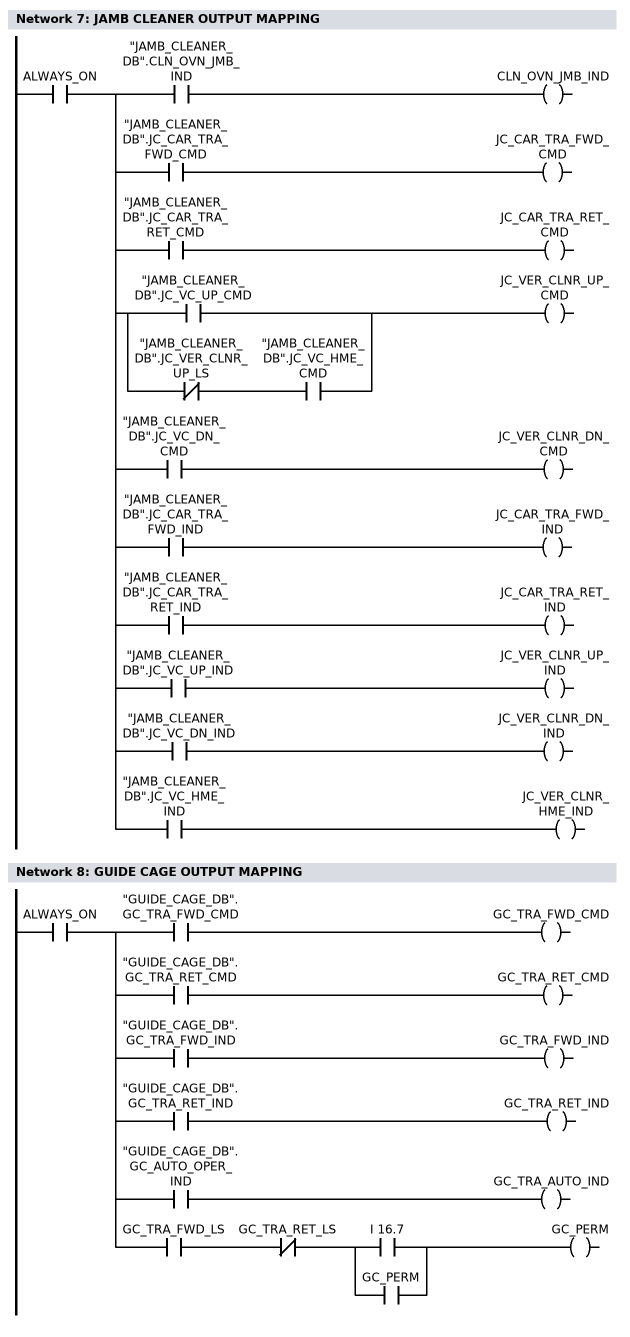
[picture p24: OUTPUT_MAPPING networks 7-8]
NETWORK
TITLE = JAMB CLEANER OUTPUT MAPPING
//JAMB CLEANER 
//
      A     "ALWAYS_ON";
      =     L 0.0;
      A     L 0.0;
      A     "JAMB_CLEANER_DB".CLN_OVN_JMB_IND;
      =     "CLN_OVN_JMB_IND";
      A     L 0.0;
      A     "JAMB_CLEANER_DB".JC_CAR_TRA_FWD_CMD;
      =     "JC_CAR_TRA_FWD_CMD";
      A     L 0.0;
      A     "JAMB_CLEANER_DB".JC_CAR_TRA_RET_CMD;
      =     "JC_CAR_TRA_RET_CMD";
      A     L 0.0;
      A(;
      O     "JAMB_CLEANER_DB".JC_VC_UP_CMD;
      O;
      AN    "JAMB_CLEANER_DB".JC_VER_CLNR_UP_LS;
      A     "JAMB_CLEANER_DB".JC_VC_HME_CMD;
      );
      =     "JC_VER_CLNR_UP_CMD";
      A     L 0.0;
      A     "JAMB_CLEANER_DB".JC_VC_DN_CMD;
      =     "JC_VER_CLNR_DN_CMD";
      A     L 0.0;
      A     "JAMB_CLEANER_DB".JC_CAR_TRA_FWD_IND;
      =     "JC_CAR_TRA_FWD_IND";
      A     L 0.0;
      A     "JAMB_CLEANER_DB".JC_CAR_TRA_RET_IND;
      =     "JC_CAR_TRA_RET_IND";
      A     L 0.0;
      A     "JAMB_CLEANER_DB".JC_VC_UP_IND;
      =     "JC_VER_CLNR_UP_IND";
      A     L 0.0;
      A     "JAMB_CLEANER_DB".JC_VC_DN_IND;
      =     "JC_VER_CLNR_DN_IND";
      A     L 0.0;
      A     "JAMB_CLEANER_DB".JC_VC_HME_IND;
      =     "JC_VER_CLNR_HME_IND";
NETWORK
TITLE = GUIDE CAGE OUTPUT MAPPING
      A     "ALWAYS_ON";
      =     L 0.0;
      A     L 0.0;
      A     "GUIDE_CAGE_DB".GC_TRA_FWD_CMD;
      =     "GC_TRA_FWD_CMD";
      A     L 0.0;
      A     "GUIDE_CAGE_DB".GC_TRA_RET_CMD;
      =     "GC_TRA_RET_CMD";
      A     L 0.0;
      A     "GUIDE_CAGE_DB".GC_TRA_FWD_IND;
      =     "GC_TRA_FWD_IND";
      A     L 0.0;
      A     "GUIDE_CAGE_DB".GC_TRA_RET_IND;
      =     "GC_TRA_RET_IND";
      A     L 0.0;
      A     "GUIDE_CAGE_DB".GC_AUTO_OPER_IND;
      =     "GC_TRA_AUTO_IND";
      A     L 0.0;
      A     "GC_TRA_FWD_LS";
      AN    "GC_TRA_RET_LS";
      A(;
      O     I 16.7;
      O     "GC_PERM";
      );
      =     "GC_PERM";
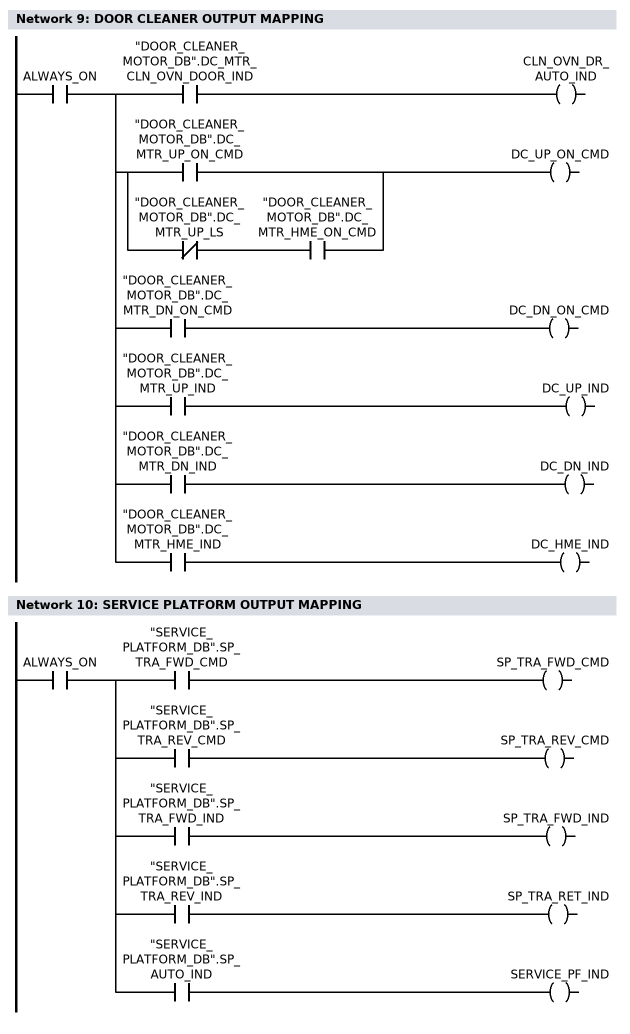
NETWORK
TITLE = DOOR CLEANER OUTPUT MAPPING
      A     "ALWAYS_ON";
      =     L 0.0;
      A     L 0.0;
      A     "DOOR_CLEANER_MOTOR_DB".DC_MTR_CLN_OVN_DOOR_IND;
      =     "CLN_OVN_DR_AUTO_IND";
      A     L 0.0;
      A(;
      O     "DOOR_CLEANER_MOTOR_DB".DC_MTR_UP_ON_CMD;
      O;
      AN    "DOOR_CLEANER_MOTOR_DB".DC_MTR_UP_LS;
      A     "DOOR_CLEANER_MOTOR_DB".DC_MTR_HME_ON_CMD;
      );
      =     "DC_UP_ON_CMD";
      A     L 0.0;
      A     "DOOR_CLEANER_MOTOR_DB".DC_MTR_DN_ON_CMD;
      =     "DC_DN_ON_CMD";
      A     L 0.0;
      A     "DOOR_CLEANER_MOTOR_DB".DC_MTR_UP_IND;
      =     "DC_UP_IND";
      A     L 0.0;
      A     "DOOR_CLEANER_MOTOR_DB".DC_MTR_DN_IND;
      =     "DC_DN_IND";
      A     L 0.0;
      A     "DOOR_CLEANER_MOTOR_DB".DC_MTR_HME_IND;
      =     "DC_HME_IND";
NETWORK
TITLE = SERVICE PLATFORM OUTPUT MAPPING
      A     "ALWAYS_ON";
      =     L 0.0;
      A     L 0.0;
      A     "SERVICE_PLATFORM_DB".SP_TRA_FWD_CMD;
      =     "SP_TRA_FWD_CMD";
      A     L 0.0;
      A     "SERVICE_PLATFORM_DB".SP_TRA_REV_CMD;
      =     "SP_TRA_REV_CMD";
      A     L 0.0;
      A     "SERVICE_PLATFORM_DB".SP_TRA_FWD_IND;
      =     "SP_TRA_FWD_IND";
      A     L 0.0;
      A     "SERVICE_PLATFORM_DB".SP_TRA_REV_IND;
      =     "SP_TRA_RET_IND";
      A     L 0.0;
      A     "SERVICE_PLATFORM_DB".SP_AUTO_IND;
      =     "SERVICE_PF_IND";
END_FUNCTION

FUNCTION "MAIN_POWER" : VOID	// FC 3
AUTHOR : Kamillas
VERSION : 0.1
BEGIN
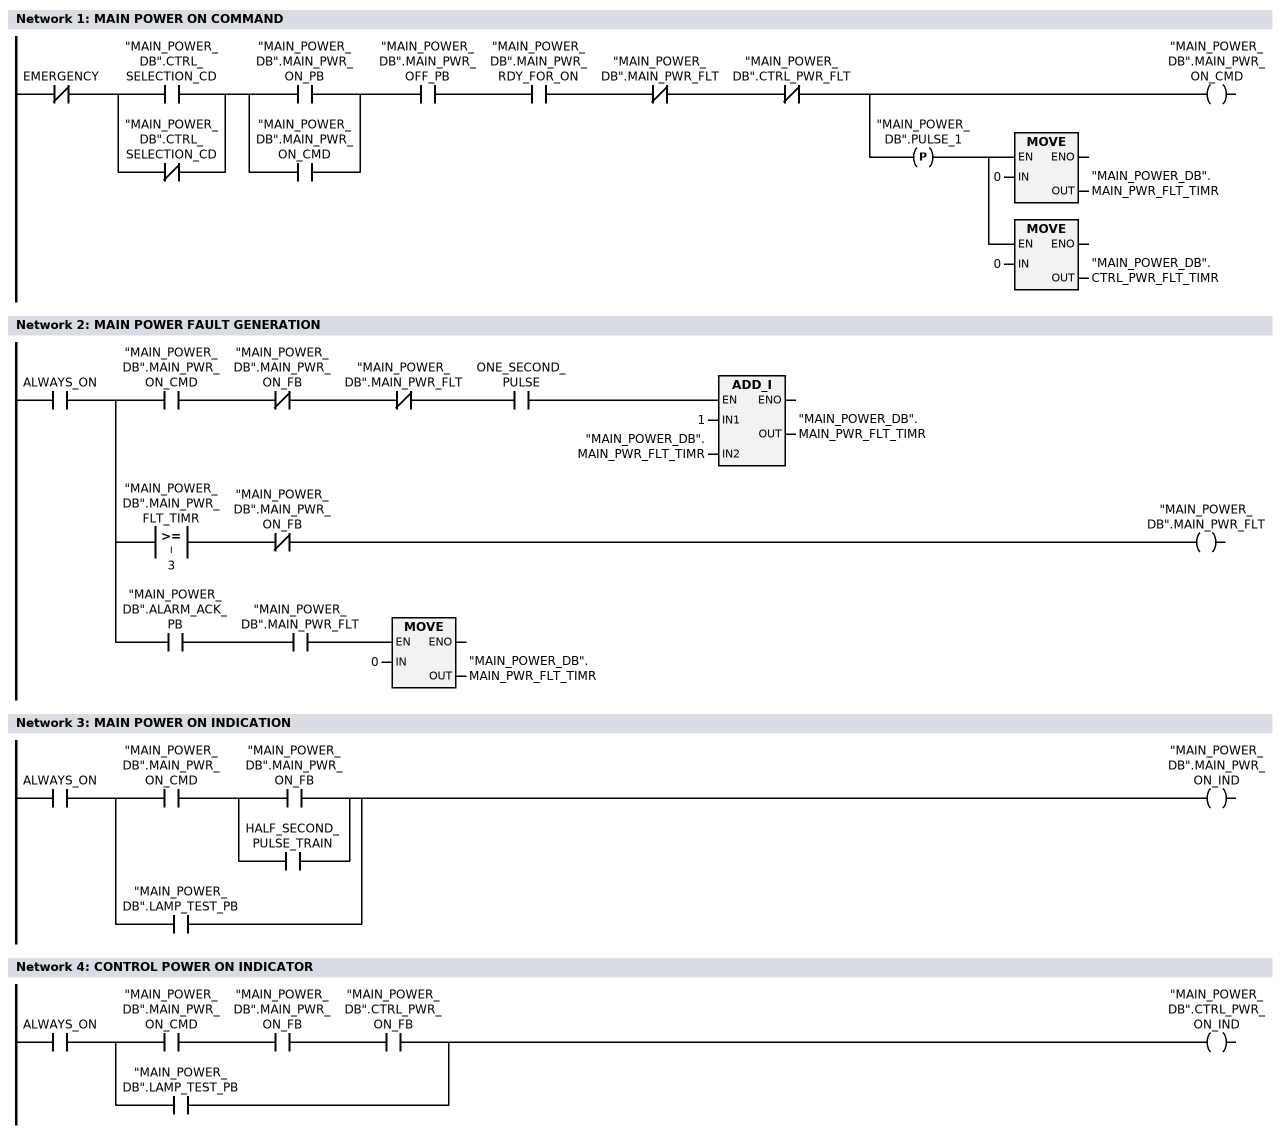
NETWORK
TITLE = MAIN POWER ON COMMAND
      AN    "EMERGENCY";
      A(;
      O     "MAIN_POWER_DB".CTRL_SELECTION_CD;
      ON    "MAIN_POWER_DB".CTRL_SELECTION_CD;
      );
      A(;
      O     "MAIN_POWER_DB".MAIN_PWR_ON_PB;
      O     "MAIN_POWER_DB".MAIN_PWR_ON_CMD;
      );
      A     "MAIN_POWER_DB".MAIN_PWR_OFF_PB;
      A     "MAIN_POWER_DB".MAIN_PWR_RDY_FOR_ON;
      AN    "MAIN_POWER_DB".MAIN_PWR_FLT;
      AN    "MAIN_POWER_DB".CTRL_PWR_FLT;
      =     L 0.0;
      A     L 0.0;
      BLD   102;
      =     "MAIN_POWER_DB".MAIN_PWR_ON_CMD;
      A     L 0.0;
      FP    "MAIN_POWER_DB".PULSE_1;
      =     L 0.1;
      A     L 0.1;
      JNB   _001;
      L     0;
      T     "MAIN_POWER_DB".MAIN_PWR_FLT_TIMR;
_001: NOP   0;
      A     L 0.1;
      JNB   _002;
      L     0;
      T     "MAIN_POWER_DB".CTRL_PWR_FLT_TIMR;
_002: NOP   0;
NETWORK
TITLE = MAIN POWER FAULT GENERATION
      A     "ALWAYS_ON";
      =     L 0.0;
      A     L 0.0;
      A     "MAIN_POWER_DB".MAIN_PWR_ON_CMD;
      AN    "MAIN_POWER_DB".MAIN_PWR_ON_FB;
      AN    "MAIN_POWER_DB".MAIN_PWR_FLT;
      A     "ONE_SECOND_PULSE";
      JNB   _003;
      L     1;
      L     "MAIN_POWER_DB".MAIN_PWR_FLT_TIMR;
      +I;
      T     "MAIN_POWER_DB".MAIN_PWR_FLT_TIMR;
_003: NOP   0;
      A     L 0.0;
      A(;
      L     "MAIN_POWER_DB".MAIN_PWR_FLT_TIMR;
      L     3;
      >=I;
      );
      AN    "MAIN_POWER_DB".MAIN_PWR_ON_FB;
      =     "MAIN_POWER_DB".MAIN_PWR_FLT;
      A     L 0.0;
      A     "MAIN_POWER_DB".ALARM_ACK_PB;
      A     "MAIN_POWER_DB".MAIN_PWR_FLT;
      JNB   _004;
      L     0;
      T     "MAIN_POWER_DB".MAIN_PWR_FLT_TIMR;
_004: NOP   0;
NETWORK
TITLE = MAIN POWER ON INDICATION
      A     "ALWAYS_ON";
      A(;
      A     "MAIN_POWER_DB".MAIN_PWR_ON_CMD;
      A(;
      O     "MAIN_POWER_DB".MAIN_PWR_ON_FB;
      O     "HALF_SECOND_PULSE_TRAIN";
      );
      O     "MAIN_POWER_DB".LAMP_TEST_PB;
      );
      =     "MAIN_POWER_DB".MAIN_PWR_ON_IND;
NETWORK
TITLE = CONTROL POWER ON INDICATOR
      A     "ALWAYS_ON";
      A(;
      A     "MAIN_POWER_DB".MAIN_PWR_ON_CMD;
      A     "MAIN_POWER_DB".MAIN_PWR_ON_FB;
      A     "MAIN_POWER_DB".CTRL_PWR_ON_FB;
      O     "MAIN_POWER_DB".LAMP_TEST_PB;
      );
      =     "MAIN_POWER_DB".CTRL_PWR_ON_IND;
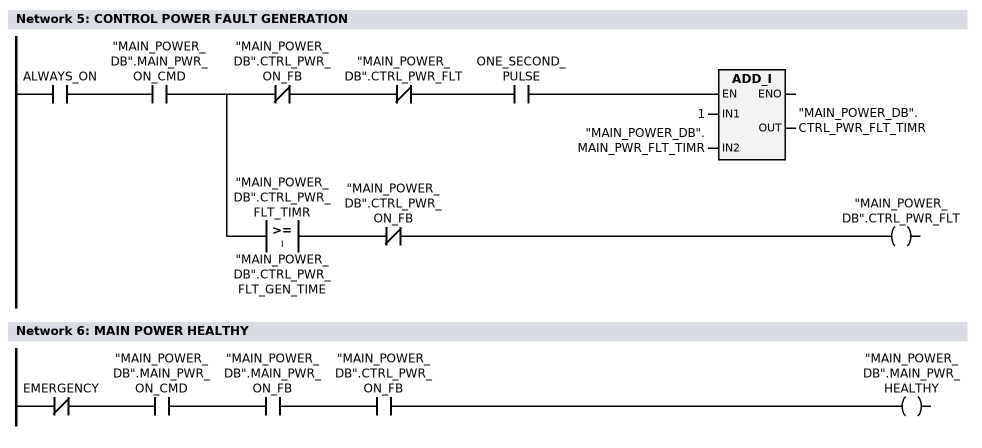
NETWORK
TITLE = CONTROL POWER FAULT GENERATION
      A     "ALWAYS_ON";
      A     "MAIN_POWER_DB".MAIN_PWR_ON_CMD;
      =     L 0.0;
      A     L 0.0;
      AN    "MAIN_POWER_DB".CTRL_PWR_ON_FB;
      AN    "MAIN_POWER_DB".CTRL_PWR_FLT;
      A     "ONE_SECOND_PULSE";
      JNB   _005;
      L     1;
      L     "MAIN_POWER_DB".MAIN_PWR_FLT_TIMR;
      +I;
      T     "MAIN_POWER_DB".CTRL_PWR_FLT_TIMR;
_005: NOP   0;
      A     L 0.0;
      A(;
      L     "MAIN_POWER_DB".CTRL_PWR_FLT_TIMR;
      L     "MAIN_POWER_DB".CTRL_PWR_FLT_GEN_TIME;
      >=I;
      );
      AN    "MAIN_POWER_DB".CTRL_PWR_ON_FB;
      =     "MAIN_POWER_DB".CTRL_PWR_FLT;
NETWORK
TITLE = MAIN POWER HEALTHY 
      AN    "EMERGENCY";
      A     "MAIN_POWER_DB".MAIN_PWR_ON_CMD;
      A     "MAIN_POWER_DB".MAIN_PWR_ON_FB;
      A     "MAIN_POWER_DB".CTRL_PWR_ON_FB;
      =     "MAIN_POWER_DB".MAIN_PWR_HEALTHY;
END_FUNCTION

FUNCTION "HYDRAULIC_SYSTEM" : VOID	// FC 4
AUTHOR : Kamillas
VERSION : 0.1
BEGIN
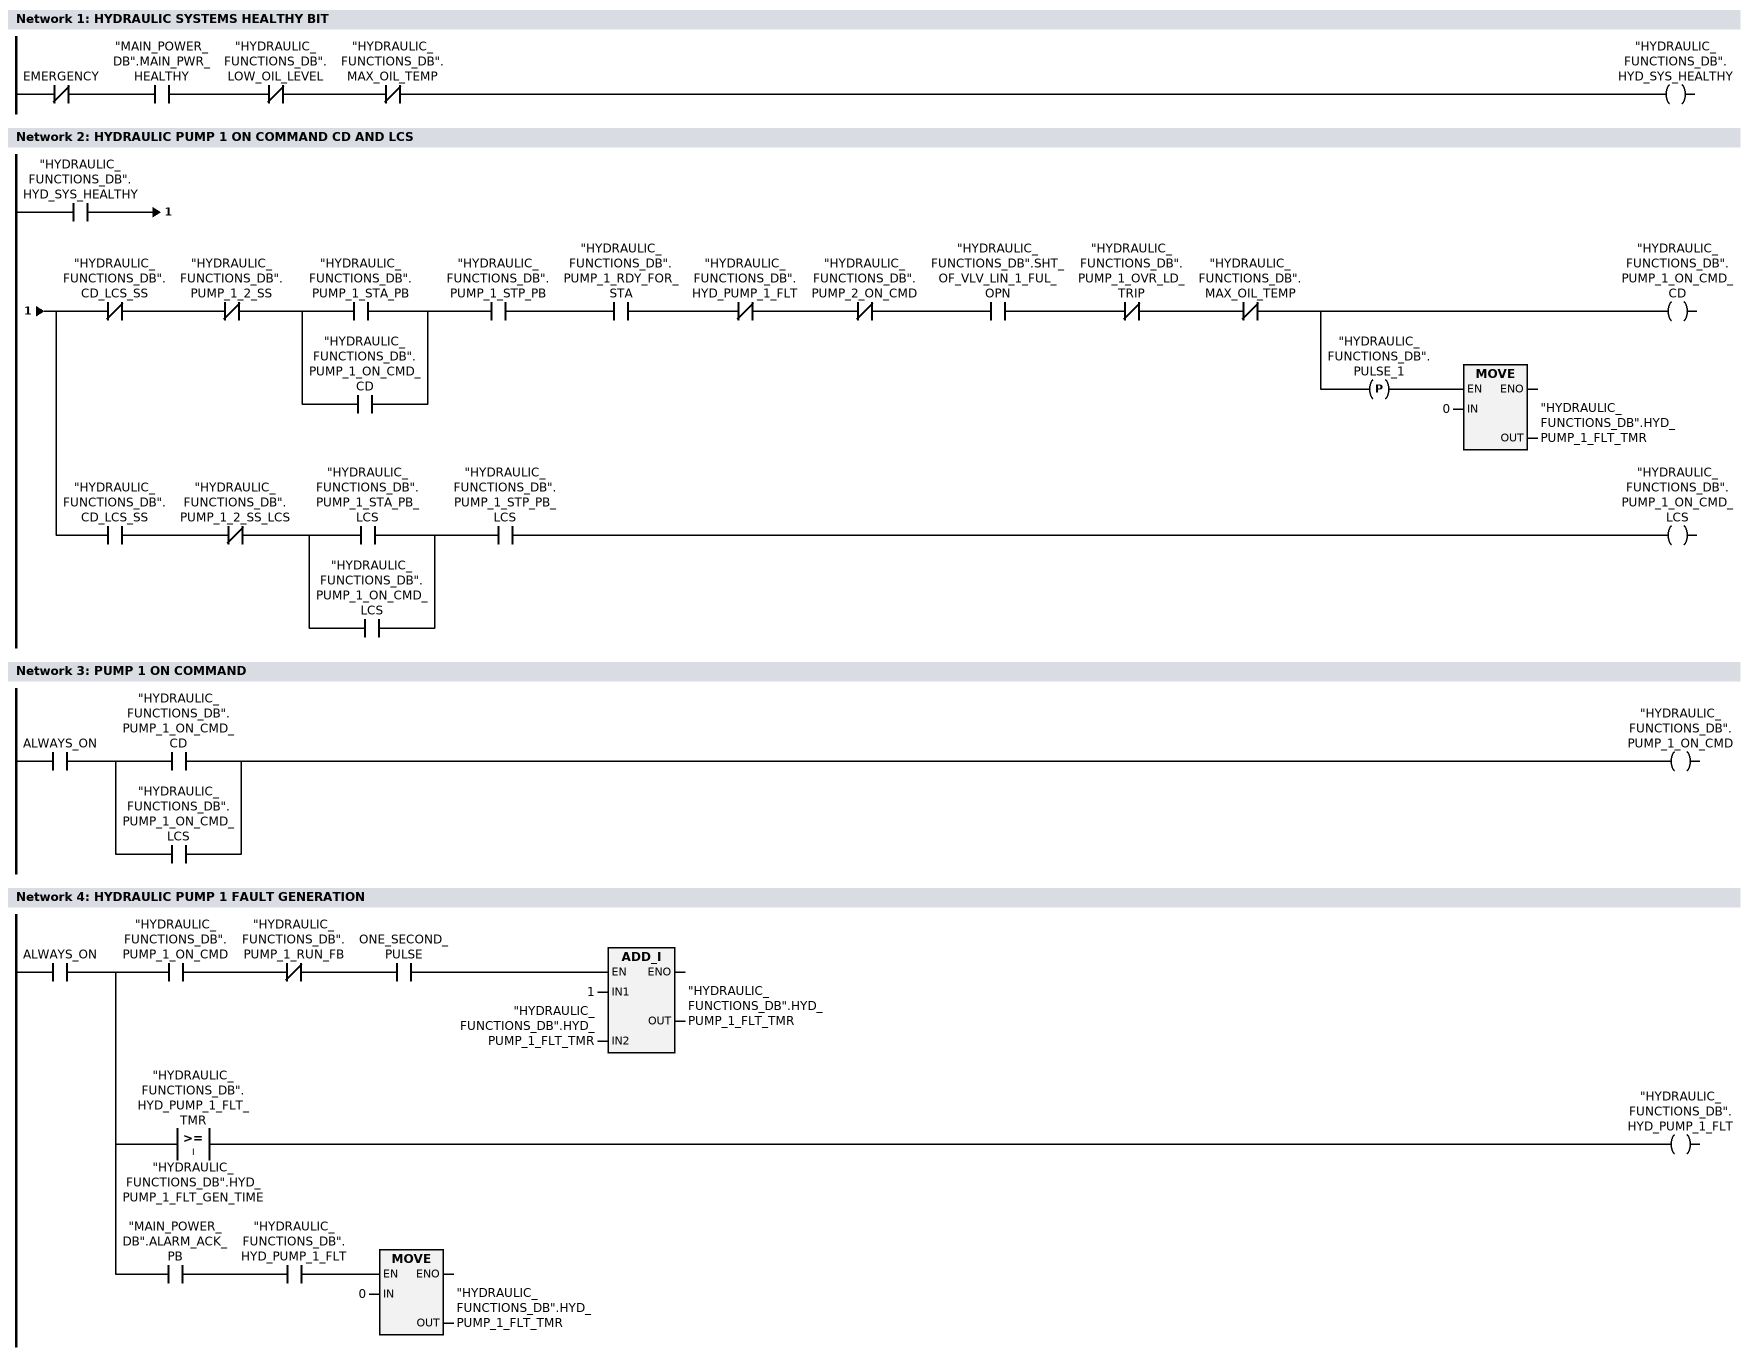
NETWORK
TITLE = HYDRAULIC SYSTEMS HEALTHY BIT
      AN    "EMERGENCY";
      A     "MAIN_POWER_DB".MAIN_PWR_HEALTHY;
      AN    "HYDRAULIC_FUNCTIONS_DB".LOW_OIL_LEVEL;
      AN    "HYDRAULIC_FUNCTIONS_DB".MAX_OIL_TEMP;
      =     "HYDRAULIC_FUNCTIONS_DB".HYD_SYS_HEALTHY;
NETWORK
TITLE = HYDRAULIC PUMP 1 ON COMMAND CD AND LCS
      A     "HYDRAULIC_FUNCTIONS_DB".HYD_SYS_HEALTHY;
      =     L 0.0;
      A     L 0.0;
      AN    "HYDRAULIC_FUNCTIONS_DB".CD_LCS_SS;
      AN    "HYDRAULIC_FUNCTIONS_DB".PUMP_1_2_SS;
      A(;
      O     "HYDRAULIC_FUNCTIONS_DB".PUMP_1_STA_PB;
      O     "HYDRAULIC_FUNCTIONS_DB".PUMP_1_ON_CMD_CD;
      );
      A     "HYDRAULIC_FUNCTIONS_DB".PUMP_1_STP_PB;
      A     "HYDRAULIC_FUNCTIONS_DB".PUMP_1_RDY_FOR_STA;
      AN    "HYDRAULIC_FUNCTIONS_DB".HYD_PUMP_1_FLT;
      AN    "HYDRAULIC_FUNCTIONS_DB".PUMP_2_ON_CMD;
      A     "HYDRAULIC_FUNCTIONS_DB".SHT_OF_VLV_LIN_1_FUL_OPN;
      AN    "HYDRAULIC_FUNCTIONS_DB".PUMP_1_OVR_LD_TRIP;
      AN    "HYDRAULIC_FUNCTIONS_DB".MAX_OIL_TEMP;
      =     L 0.1;
      A     L 0.1;
      BLD   102;
      =     "HYDRAULIC_FUNCTIONS_DB".PUMP_1_ON_CMD_CD;
      A     L 0.1;
      FP    "HYDRAULIC_FUNCTIONS_DB".PULSE_1;
      JNB   _001;
      L     0;
      T     "HYDRAULIC_FUNCTIONS_DB".HYD_PUMP_1_FLT_TMR;
_001: NOP   0;
      A     L 0.0;
      A     "HYDRAULIC_FUNCTIONS_DB".CD_LCS_SS;
      AN    "HYDRAULIC_FUNCTIONS_DB".PUMP_1_2_SS_LCS;
      A(;
      O     "HYDRAULIC_FUNCTIONS_DB".PUMP_1_STA_PB_LCS;
      O     "HYDRAULIC_FUNCTIONS_DB".PUMP_1_ON_CMD_LCS;
      );
      A     "HYDRAULIC_FUNCTIONS_DB".PUMP_1_STP_PB_LCS;
      =     "HYDRAULIC_FUNCTIONS_DB".PUMP_1_ON_CMD_LCS;
NETWORK
TITLE = PUMP 1 ON COMMAND
      A     "ALWAYS_ON";
      A(;
      O     "HYDRAULIC_FUNCTIONS_DB".PUMP_1_ON_CMD_CD;
      O     "HYDRAULIC_FUNCTIONS_DB".PUMP_1_ON_CMD_LCS;
      );
      =     "HYDRAULIC_FUNCTIONS_DB".PUMP_1_ON_CMD;
NETWORK
TITLE = HYDRAULIC PUMP 1 FAULT GENERATION
      A     "ALWAYS_ON";
      =     L 0.0;
      A     L 0.0;
      A     "HYDRAULIC_FUNCTIONS_DB".PUMP_1_ON_CMD;
      AN    "HYDRAULIC_FUNCTIONS_DB".PUMP_1_RUN_FB;
      A     "ONE_SECOND_PULSE";
      JNB   _002;
      L     1;
      L     "HYDRAULIC_FUNCTIONS_DB".HYD_PUMP_1_FLT_TMR;
      +I;
      T     "HYDRAULIC_FUNCTIONS_DB".HYD_PUMP_1_FLT_TMR;
_002: NOP   0;
      A     L 0.0;
      A(;
      L     "HYDRAULIC_FUNCTIONS_DB".HYD_PUMP_1_FLT_TMR;
      L     "HYDRAULIC_FUNCTIONS_DB".HYD_PUMP_1_FLT_GEN_TIME;
      >=I;
      );
      =     "HYDRAULIC_FUNCTIONS_DB".HYD_PUMP_1_FLT;
      A     L 0.0;
      A     "MAIN_POWER_DB".ALARM_ACK_PB;
      A     "HYDRAULIC_FUNCTIONS_DB".HYD_PUMP_1_FLT;
      JNB   _003;
      L     0;
      T     "HYDRAULIC_FUNCTIONS_DB".HYD_PUMP_1_FLT_TMR;
_003: NOP   0;
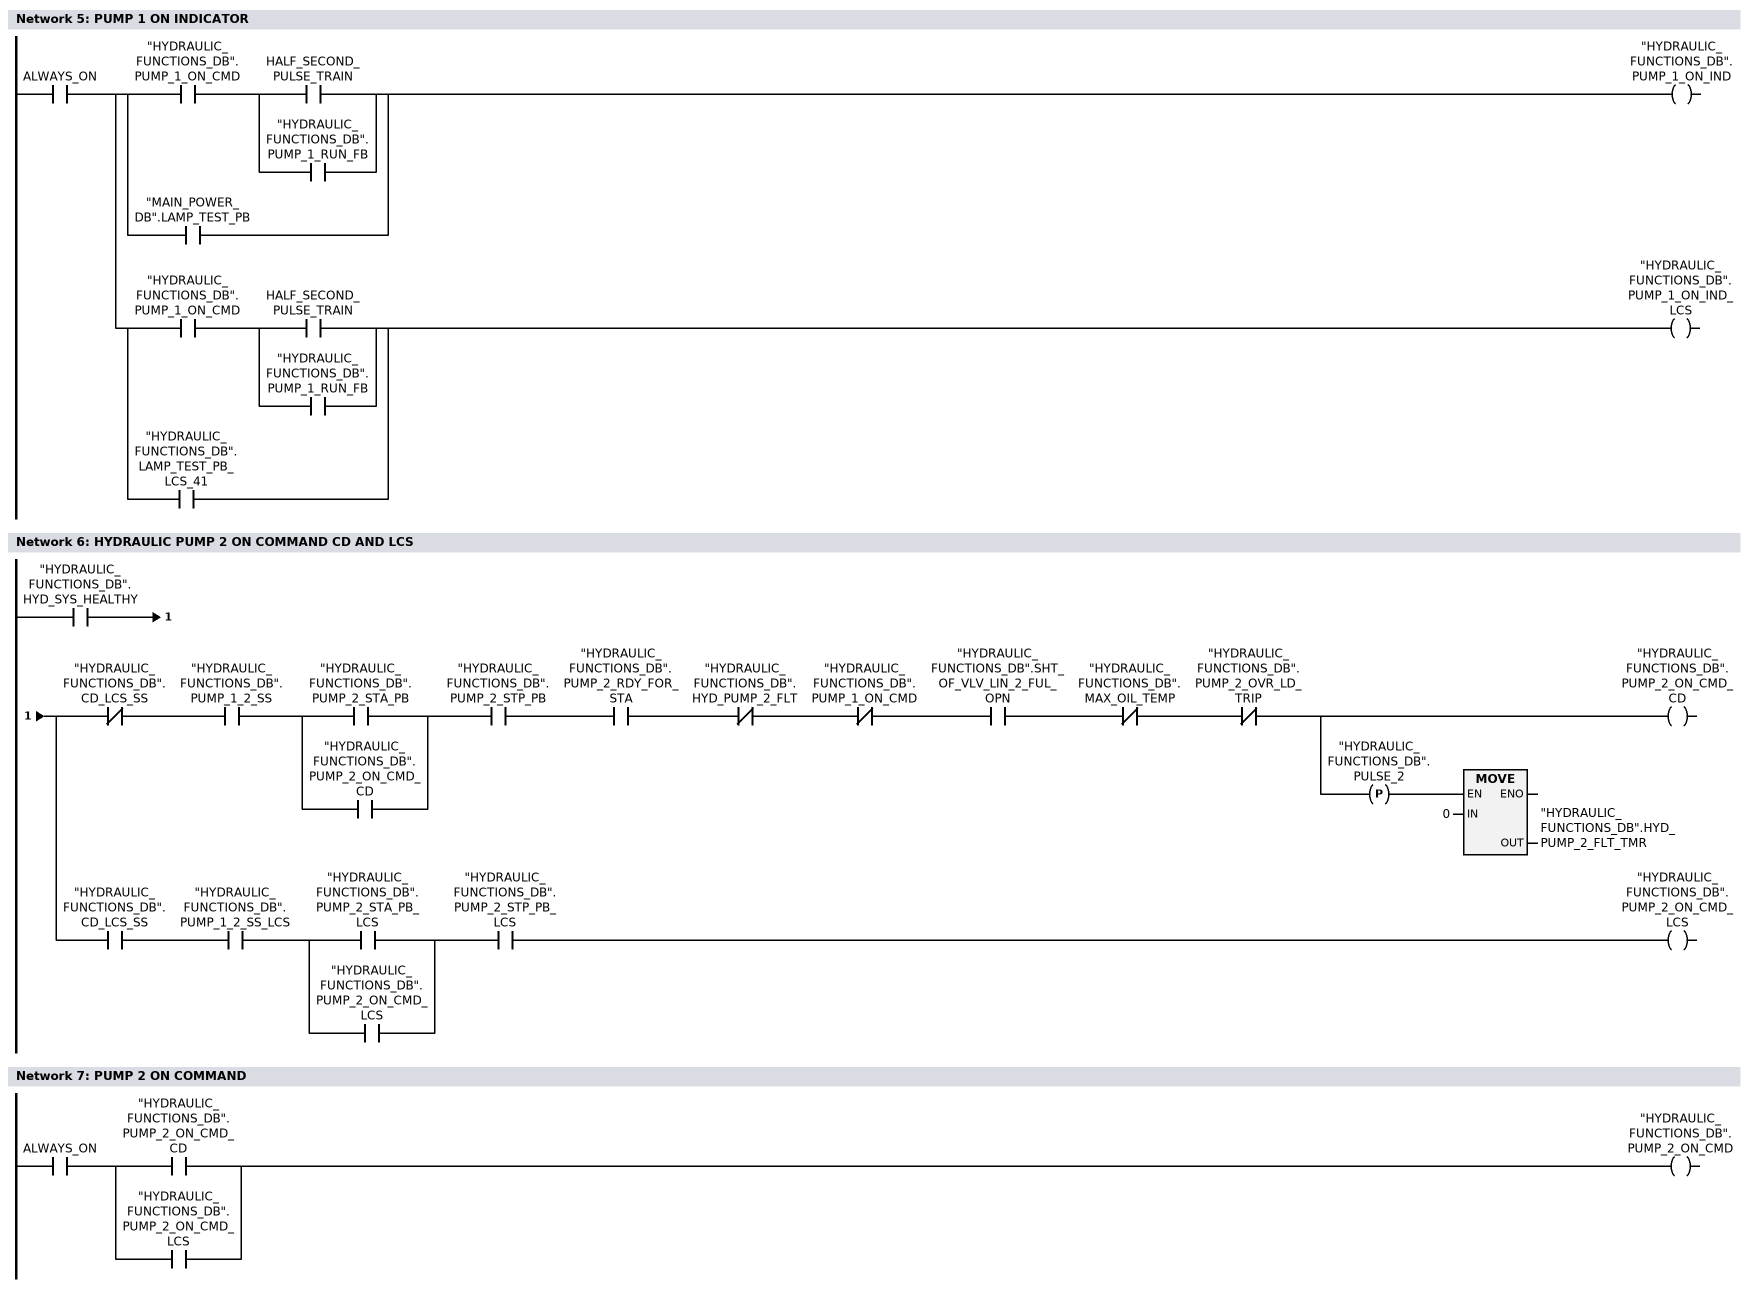
NETWORK
TITLE = PUMP 1 ON INDICATOR
      A     "ALWAYS_ON";
      =     L 0.0;
      A     L 0.0;
      A(;
      A     "HYDRAULIC_FUNCTIONS_DB".PUMP_1_ON_CMD;
      A(;
      O     "HALF_SECOND_PULSE_TRAIN";
      O     "HYDRAULIC_FUNCTIONS_DB".PUMP_1_RUN_FB;
      );
      O     "MAIN_POWER_DB".LAMP_TEST_PB;
      );
      =     "HYDRAULIC_FUNCTIONS_DB".PUMP_1_ON_IND;
      A     L 0.0;
      A(;
      A     "HYDRAULIC_FUNCTIONS_DB".PUMP_1_ON_CMD;
      A(;
      O     "HALF_SECOND_PULSE_TRAIN";
      O     "HYDRAULIC_FUNCTIONS_DB".PUMP_1_RUN_FB;
      );
      O     "HYDRAULIC_FUNCTIONS_DB".LAMP_TEST_PB_LCS_41;
      );
      =     "HYDRAULIC_FUNCTIONS_DB".PUMP_1_ON_IND_LCS;
NETWORK
TITLE = HYDRAULIC PUMP 2 ON COMMAND CD AND LCS
      A     "HYDRAULIC_FUNCTIONS_DB".HYD_SYS_HEALTHY;
      =     L 0.0;
      A     L 0.0;
      AN    "HYDRAULIC_FUNCTIONS_DB".CD_LCS_SS;
      A     "HYDRAULIC_FUNCTIONS_DB".PUMP_1_2_SS;
      A(;
      O     "HYDRAULIC_FUNCTIONS_DB".PUMP_2_STA_PB;
      O     "HYDRAULIC_FUNCTIONS_DB".PUMP_2_ON_CMD_CD;
      );
      A     "HYDRAULIC_FUNCTIONS_DB".PUMP_2_STP_PB;
      A     "HYDRAULIC_FUNCTIONS_DB".PUMP_2_RDY_FOR_STA;
      AN    "HYDRAULIC_FUNCTIONS_DB".HYD_PUMP_2_FLT;
      AN    "HYDRAULIC_FUNCTIONS_DB".PUMP_1_ON_CMD;
      A     "HYDRAULIC_FUNCTIONS_DB".SHT_OF_VLV_LIN_2_FUL_OPN;
      AN    "HYDRAULIC_FUNCTIONS_DB".MAX_OIL_TEMP;
      AN    "HYDRAULIC_FUNCTIONS_DB".PUMP_2_OVR_LD_TRIP;
      =     L 0.1;
      A     L 0.1;
      BLD   102;
      =     "HYDRAULIC_FUNCTIONS_DB".PUMP_2_ON_CMD_CD;
      A     L 0.1;
      FP    "HYDRAULIC_FUNCTIONS_DB".PULSE_2;
      JNB   _004;
      L     0;
      T     "HYDRAULIC_FUNCTIONS_DB".HYD_PUMP_2_FLT_TMR;
_004: NOP   0;
      A     L 0.0;
      A     "HYDRAULIC_FUNCTIONS_DB".CD_LCS_SS;
      A     "HYDRAULIC_FUNCTIONS_DB".PUMP_1_2_SS_LCS;
      A(;
      O     "HYDRAULIC_FUNCTIONS_DB".PUMP_2_STA_PB_LCS;
      O     "HYDRAULIC_FUNCTIONS_DB".PUMP_2_ON_CMD_LCS;
      );
      A     "HYDRAULIC_FUNCTIONS_DB".PUMP_2_STP_PB_LCS;
      =     "HYDRAULIC_FUNCTIONS_DB".PUMP_2_ON_CMD_LCS;
NETWORK
TITLE = PUMP 2 ON COMMAND
      A     "ALWAYS_ON";
      A(;
      O     "HYDRAULIC_FUNCTIONS_DB".PUMP_2_ON_CMD_CD;
      O     "HYDRAULIC_FUNCTIONS_DB".PUMP_2_ON_CMD_LCS;
      );
      =     "HYDRAULIC_FUNCTIONS_DB".PUMP_2_ON_CMD;
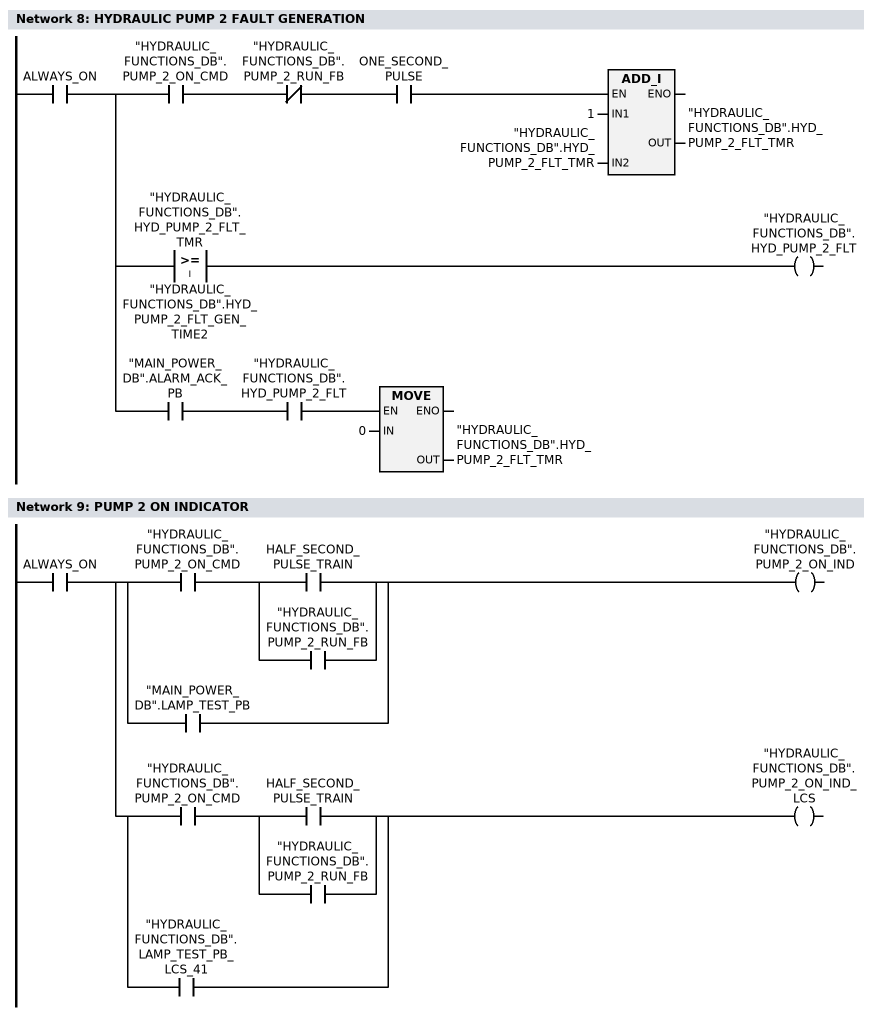
NETWORK
TITLE = HYDRAULIC PUMP 2 FAULT GENERATION
      A     "ALWAYS_ON";
      =     L 0.0;
      A     L 0.0;
      A     "HYDRAULIC_FUNCTIONS_DB".PUMP_2_ON_CMD;
      AN    "HYDRAULIC_FUNCTIONS_DB".PUMP_2_RUN_FB;
      A     "ONE_SECOND_PULSE";
      JNB   _005;
      L     1;
      L     "HYDRAULIC_FUNCTIONS_DB".HYD_PUMP_2_FLT_TMR;
      +I;
      T     "HYDRAULIC_FUNCTIONS_DB".HYD_PUMP_2_FLT_TMR;
_005: NOP   0;
      A     L 0.0;
      A(;
      L     "HYDRAULIC_FUNCTIONS_DB".HYD_PUMP_2_FLT_TMR;
      L     "HYDRAULIC_FUNCTIONS_DB".HYD_PUMP_2_FLT_GEN_TIME2;
      >=I;
      );
      =     "HYDRAULIC_FUNCTIONS_DB".HYD_PUMP_2_FLT;
      A     L 0.0;
      A     "MAIN_POWER_DB".ALARM_ACK_PB;
      A     "HYDRAULIC_FUNCTIONS_DB".HYD_PUMP_2_FLT;
      JNB   _006;
      L     0;
      T     "HYDRAULIC_FUNCTIONS_DB".HYD_PUMP_2_FLT_TMR;
_006: NOP   0;
NETWORK
TITLE = PUMP 2 ON INDICATOR
      A     "ALWAYS_ON";
      =     L 0.0;
      A     L 0.0;
      A(;
      A     "HYDRAULIC_FUNCTIONS_DB".PUMP_2_ON_CMD;
      A(;
      O     "HALF_SECOND_PULSE_TRAIN";
      O     "HYDRAULIC_FUNCTIONS_DB".PUMP_2_RUN_FB;
      );
      O     "MAIN_POWER_DB".LAMP_TEST_PB;
      );
      =     "HYDRAULIC_FUNCTIONS_DB".PUMP_2_ON_IND;
      A     L 0.0;
      A(;
      A     "HYDRAULIC_FUNCTIONS_DB".PUMP_2_ON_CMD;
      A(;
      O     "HALF_SECOND_PULSE_TRAIN";
      O     "HYDRAULIC_FUNCTIONS_DB".PUMP_2_RUN_FB;
      );
      O     "HYDRAULIC_FUNCTIONS_DB".LAMP_TEST_PB_LCS_41;
      );
      =     "HYDRAULIC_FUNCTIONS_DB".PUMP_2_ON_IND_LCS;
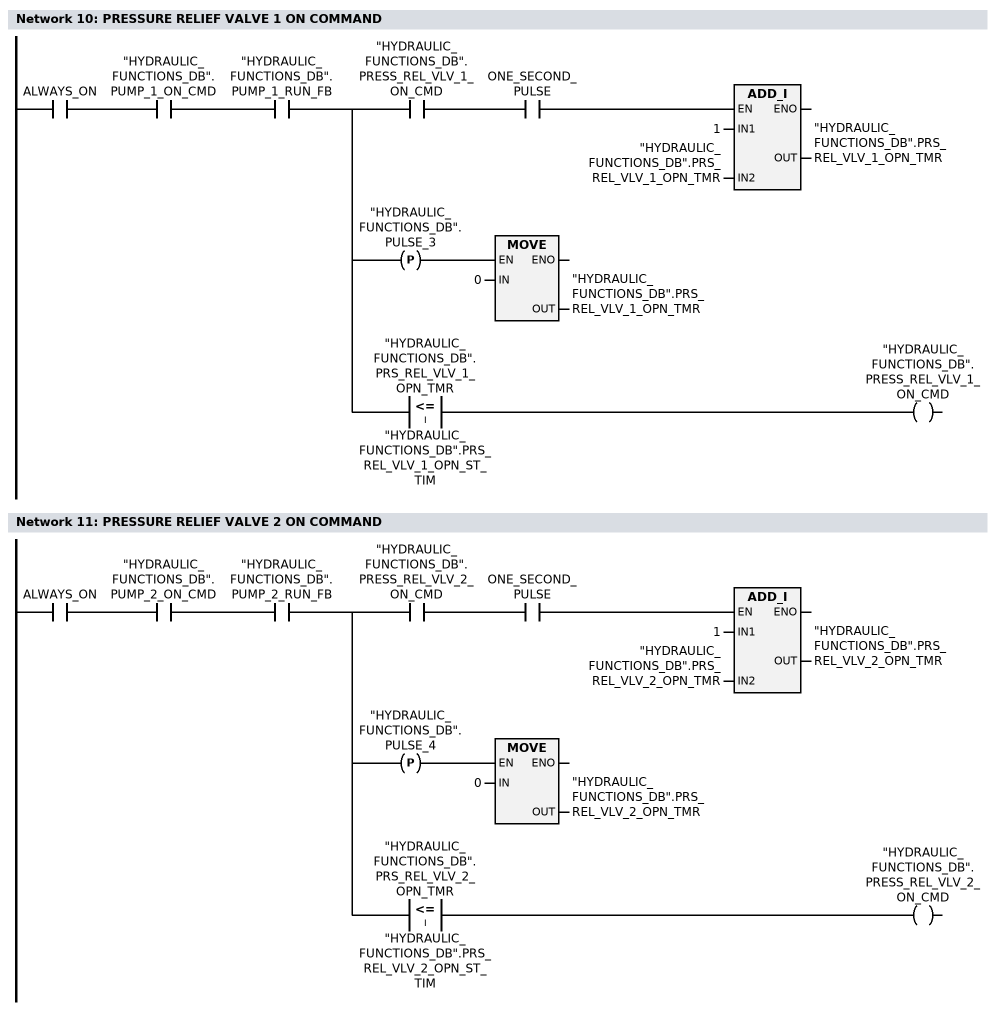
NETWORK
TITLE = PRESSURE RELIEF VALVE 1 ON COMMAND
      A     "ALWAYS_ON";
      A     "HYDRAULIC_FUNCTIONS_DB".PUMP_1_ON_CMD;
      A     "HYDRAULIC_FUNCTIONS_DB".PUMP_1_RUN_FB;
      =     L 0.0;
      A     L 0.0;
      A     "HYDRAULIC_FUNCTIONS_DB".PRESS_REL_VLV_1_ON_CMD;
      A     "ONE_SECOND_PULSE";
      JNB   _007;
      L     1;
      L     "HYDRAULIC_FUNCTIONS_DB".PRS_REL_VLV_1_OPN_TMR;
      +I;
      T     "HYDRAULIC_FUNCTIONS_DB".PRS_REL_VLV_1_OPN_TMR;
_007: NOP   0;
      A     L 0.0;
      FP    "HYDRAULIC_FUNCTIONS_DB".PULSE_3;
      JNB   _008;
      L     0;
      T     "HYDRAULIC_FUNCTIONS_DB".PRS_REL_VLV_1_OPN_TMR;
_008: NOP   0;
      A     L 0.0;
      A(;
      L     "HYDRAULIC_FUNCTIONS_DB".PRS_REL_VLV_1_OPN_TMR;
      L     "HYDRAULIC_FUNCTIONS_DB".PRS_REL_VLV_1_OPN_ST_TIM;
      <=I;
      );
      =     "HYDRAULIC_FUNCTIONS_DB".PRESS_REL_VLV_1_ON_CMD;
NETWORK
TITLE = PRESSURE RELIEF VALVE 2 ON COMMAND
      A     "ALWAYS_ON";
      A     "HYDRAULIC_FUNCTIONS_DB".PUMP_2_ON_CMD;
      A     "HYDRAULIC_FUNCTIONS_DB".PUMP_2_RUN_FB;
      =     L 0.0;
      A     L 0.0;
      A     "HYDRAULIC_FUNCTIONS_DB".PRESS_REL_VLV_2_ON_CMD;
      A     "ONE_SECOND_PULSE";
      JNB   _009;
      L     1;
      L     "HYDRAULIC_FUNCTIONS_DB".PRS_REL_VLV_2_OPN_TMR;
      +I;
      T     "HYDRAULIC_FUNCTIONS_DB".PRS_REL_VLV_2_OPN_TMR;
_009: NOP   0;
      A     L 0.0;
      FP    "HYDRAULIC_FUNCTIONS_DB".PULSE_4;
      JNB   _00a;
      L     0;
      T     "HYDRAULIC_FUNCTIONS_DB".PRS_REL_VLV_2_OPN_TMR;
_00a: NOP   0;
      A     L 0.0;
      A(;
      L     "HYDRAULIC_FUNCTIONS_DB".PRS_REL_VLV_2_OPN_TMR;
      L     "HYDRAULIC_FUNCTIONS_DB".PRS_REL_VLV_2_OPN_ST_TIM;
      <=I;
      );
      =     "HYDRAULIC_FUNCTIONS_DB".PRESS_REL_VLV_2_ON_CMD;
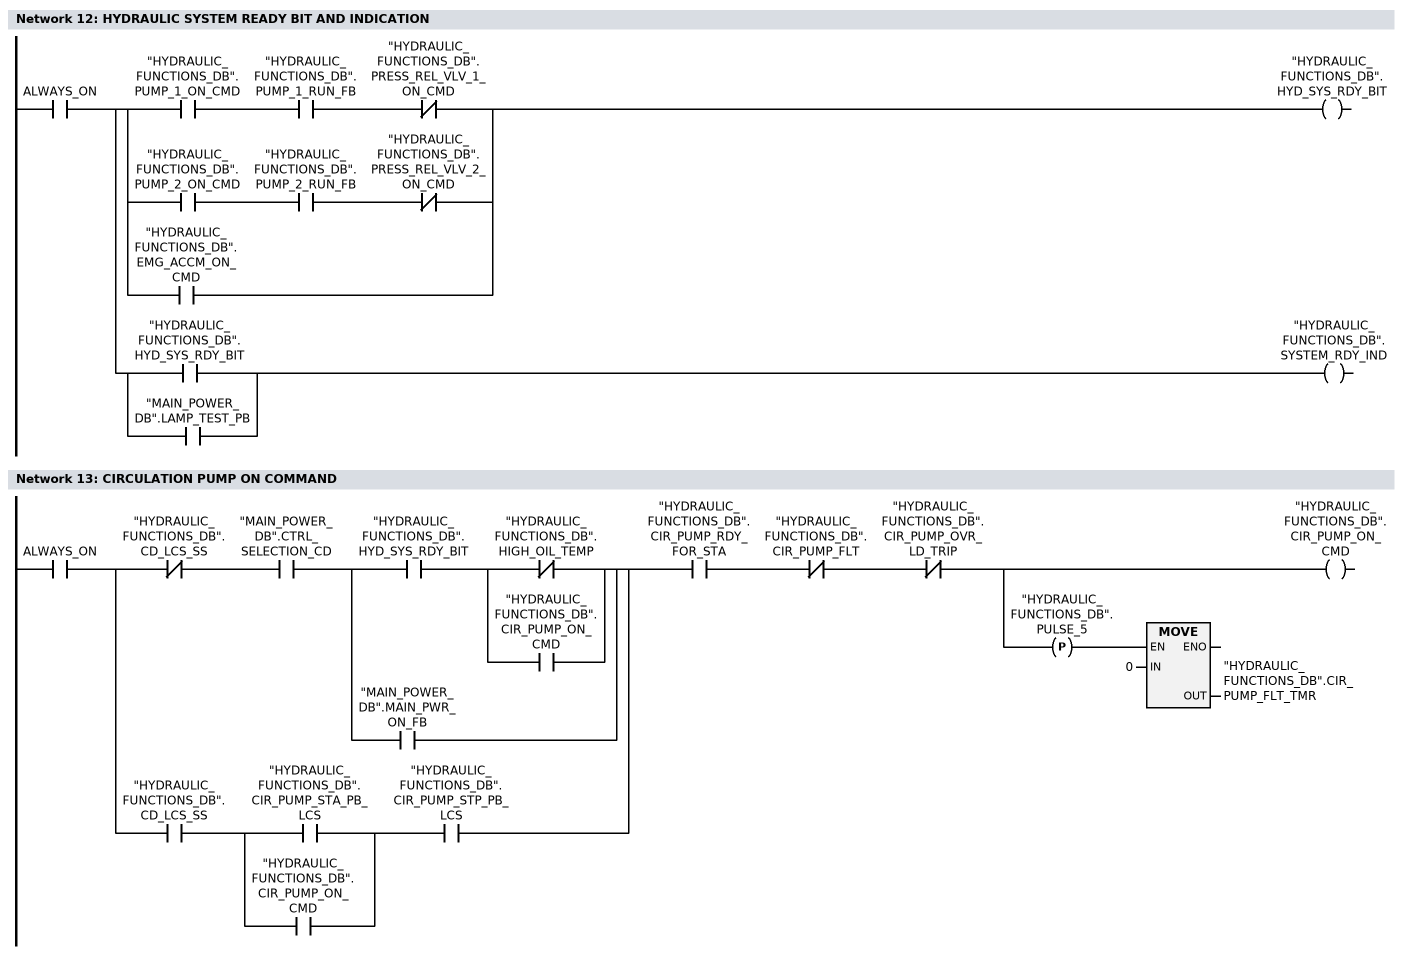
NETWORK
TITLE = HYDRAULIC SYSTEM READY BIT AND INDICATION
      A     "ALWAYS_ON";
      =     L 0.0;
      A     L 0.0;
      A(;
      A     "HYDRAULIC_FUNCTIONS_DB".PUMP_1_ON_CMD;
      A     "HYDRAULIC_FUNCTIONS_DB".PUMP_1_RUN_FB;
      AN    "HYDRAULIC_FUNCTIONS_DB".PRESS_REL_VLV_1_ON_CMD;
      O;
      A     "HYDRAULIC_FUNCTIONS_DB".PUMP_2_ON_CMD;
      A     "HYDRAULIC_FUNCTIONS_DB".PUMP_2_RUN_FB;
      AN    "HYDRAULIC_FUNCTIONS_DB".PRESS_REL_VLV_2_ON_CMD;
      O     "HYDRAULIC_FUNCTIONS_DB".EMG_ACCM_ON_CMD;
      );
      =     "HYDRAULIC_FUNCTIONS_DB".HYD_SYS_RDY_BIT;
      A     L 0.0;
      A(;
      O     "HYDRAULIC_FUNCTIONS_DB".HYD_SYS_RDY_BIT;
      O     "MAIN_POWER_DB".LAMP_TEST_PB;
      );
      =     "HYDRAULIC_FUNCTIONS_DB".SYSTEM_RDY_IND;
NETWORK
TITLE = CIRCULATION PUMP ON COMMAND
      A     "ALWAYS_ON";
      A(;
      AN    "HYDRAULIC_FUNCTIONS_DB".CD_LCS_SS;
      A     "MAIN_POWER_DB".CTRL_SELECTION_CD;
      A(;
      A     "HYDRAULIC_FUNCTIONS_DB".HYD_SYS_RDY_BIT;
      A(;
      ON    "HYDRAULIC_FUNCTIONS_DB".HIGH_OIL_TEMP;
      O     "HYDRAULIC_FUNCTIONS_DB".CIR_PUMP_ON_CMD;
      );
      O     "MAIN_POWER_DB".MAIN_PWR_ON_FB;
      );
      O;
      A     "HYDRAULIC_FUNCTIONS_DB".CD_LCS_SS;
      A(;
      O     "HYDRAULIC_FUNCTIONS_DB".CIR_PUMP_STA_PB_LCS;
      O     "HYDRAULIC_FUNCTIONS_DB".CIR_PUMP_ON_CMD;
      );
      A     "HYDRAULIC_FUNCTIONS_DB".CIR_PUMP_STP_PB_LCS;
      );
      A     "HYDRAULIC_FUNCTIONS_DB".CIR_PUMP_RDY_FOR_STA;
      AN    "HYDRAULIC_FUNCTIONS_DB".CIR_PUMP_FLT;
      AN    "HYDRAULIC_FUNCTIONS_DB".CIR_PUMP_OVR_LD_TRIP;
      =     L 0.0;
      A     L 0.0;
      BLD   102;
      =     "HYDRAULIC_FUNCTIONS_DB".CIR_PUMP_ON_CMD;
      A     L 0.0;
      FP    "HYDRAULIC_FUNCTIONS_DB".PULSE_5;
      JNB   _00b;
      L     0;
      T     "HYDRAULIC_FUNCTIONS_DB".CIR_PUMP_FLT_TMR;
_00b: NOP   0;
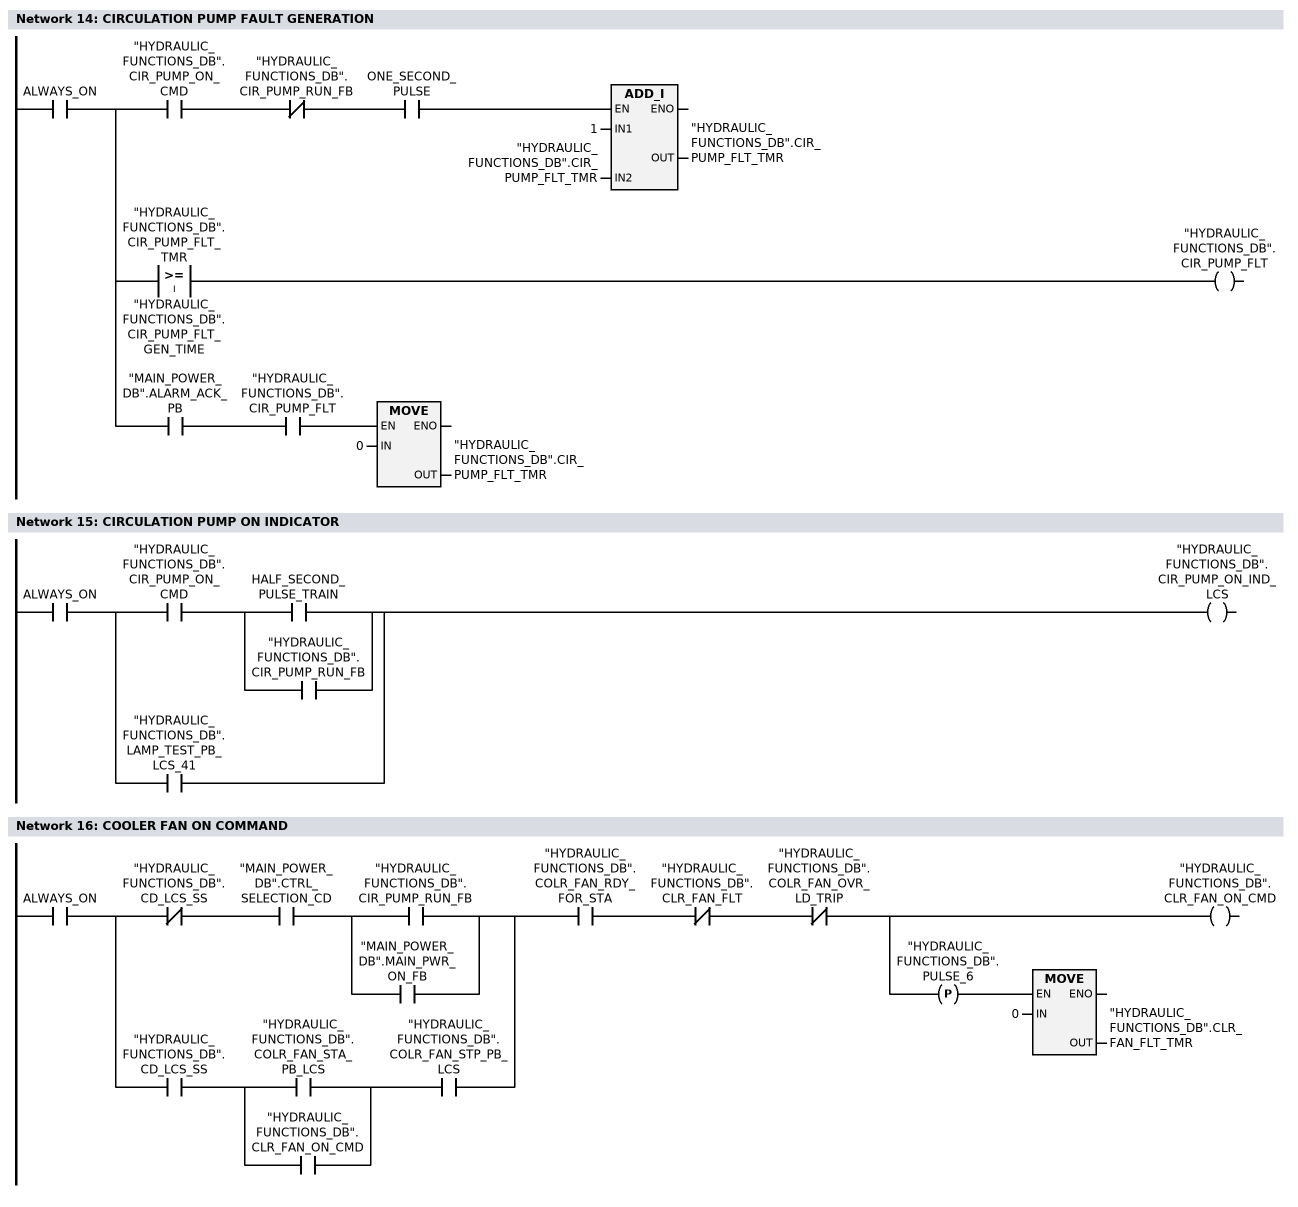
NETWORK
TITLE = CIRCULATION PUMP FAULT GENERATION
      A     "ALWAYS_ON";
      =     L 0.0;
      A     L 0.0;
      A     "HYDRAULIC_FUNCTIONS_DB".CIR_PUMP_ON_CMD;
      AN    "HYDRAULIC_FUNCTIONS_DB".CIR_PUMP_RUN_FB;
      A     "ONE_SECOND_PULSE";
      JNB   _00c;
      L     1;
      L     "HYDRAULIC_FUNCTIONS_DB".CIR_PUMP_FLT_TMR;
      +I;
      T     "HYDRAULIC_FUNCTIONS_DB".CIR_PUMP_FLT_TMR;
_00c: NOP   0;
      A     L 0.0;
      A(;
      L     "HYDRAULIC_FUNCTIONS_DB".CIR_PUMP_FLT_TMR;
      L     "HYDRAULIC_FUNCTIONS_DB".CIR_PUMP_FLT_GEN_TIME;
      >=I;
      );
      =     "HYDRAULIC_FUNCTIONS_DB".CIR_PUMP_FLT;
      A     L 0.0;
      A     "MAIN_POWER_DB".ALARM_ACK_PB;
      A     "HYDRAULIC_FUNCTIONS_DB".CIR_PUMP_FLT;
      JNB   _00d;
      L     0;
      T     "HYDRAULIC_FUNCTIONS_DB".CIR_PUMP_FLT_TMR;
_00d: NOP   0;
NETWORK
TITLE = CIRCULATION PUMP ON INDICATOR
      A     "ALWAYS_ON";
      A(;
      A     "HYDRAULIC_FUNCTIONS_DB".CIR_PUMP_ON_CMD;
      A(;
      O     "HALF_SECOND_PULSE_TRAIN";
      O     "HYDRAULIC_FUNCTIONS_DB".CIR_PUMP_RUN_FB;
      );
      O     "HYDRAULIC_FUNCTIONS_DB".LAMP_TEST_PB_LCS_41;
      );
      =     "HYDRAULIC_FUNCTIONS_DB".CIR_PUMP_ON_IND_LCS;
NETWORK
TITLE = COOLER FAN ON COMMAND
      A     "ALWAYS_ON";
      A(;
      AN    "HYDRAULIC_FUNCTIONS_DB".CD_LCS_SS;
      A     "MAIN_POWER_DB".CTRL_SELECTION_CD;
      A(;
      O     "HYDRAULIC_FUNCTIONS_DB".CIR_PUMP_RUN_FB;
      O     "MAIN_POWER_DB".MAIN_PWR_ON_FB;
      );
      O;
      A     "HYDRAULIC_FUNCTIONS_DB".CD_LCS_SS;
      A(;
      O     "HYDRAULIC_FUNCTIONS_DB".COLR_FAN_STA_PB_LCS;
      O     "HYDRAULIC_FUNCTIONS_DB".CLR_FAN_ON_CMD;
      );
      A     "HYDRAULIC_FUNCTIONS_DB".COLR_FAN_STP_PB_LCS;
      );
      A     "HYDRAULIC_FUNCTIONS_DB".COLR_FAN_RDY_FOR_STA;
      AN    "HYDRAULIC_FUNCTIONS_DB".CLR_FAN_FLT;
      AN    "HYDRAULIC_FUNCTIONS_DB".COLR_FAN_OVR_LD_TRIP;
      =     L 0.0;
      A     L 0.0;
      BLD   102;
      =     "HYDRAULIC_FUNCTIONS_DB".CLR_FAN_ON_CMD;
      A     L 0.0;
      FP    "HYDRAULIC_FUNCTIONS_DB".PULSE_6;
      JNB   _00e;
      L     0;
      T     "HYDRAULIC_FUNCTIONS_DB".CLR_FAN_FLT_TMR;
_00e: NOP   0;
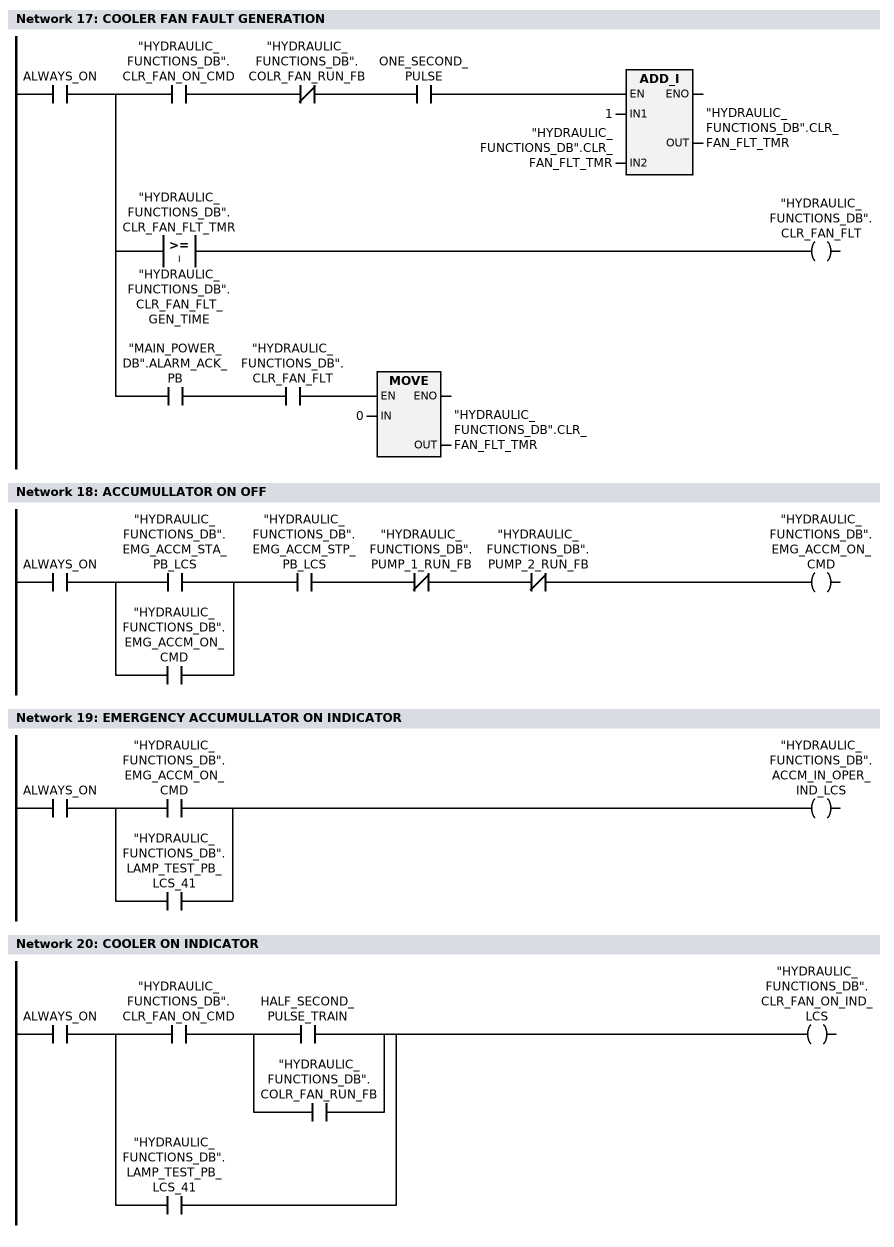
NETWORK
TITLE = COOLER FAN FAULT GENERATION
      A     "ALWAYS_ON";
      =     L 0.0;
      A     L 0.0;
      A     "HYDRAULIC_FUNCTIONS_DB".CLR_FAN_ON_CMD;
      AN    "HYDRAULIC_FUNCTIONS_DB".COLR_FAN_RUN_FB;
      A     "ONE_SECOND_PULSE";
      JNB   _00f;
      L     1;
      L     "HYDRAULIC_FUNCTIONS_DB".CLR_FAN_FLT_TMR;
      +I;
      T     "HYDRAULIC_FUNCTIONS_DB".CLR_FAN_FLT_TMR;
_00f: NOP   0;
      A     L 0.0;
      A(;
      L     "HYDRAULIC_FUNCTIONS_DB".CLR_FAN_FLT_TMR;
      L     "HYDRAULIC_FUNCTIONS_DB".CLR_FAN_FLT_GEN_TIME;
      >=I;
      );
      =     "HYDRAULIC_FUNCTIONS_DB".CLR_FAN_FLT;
      A     L 0.0;
      A     "MAIN_POWER_DB".ALARM_ACK_PB;
      A     "HYDRAULIC_FUNCTIONS_DB".CLR_FAN_FLT;
      JNB   _010;
      L     0;
      T     "HYDRAULIC_FUNCTIONS_DB".CLR_FAN_FLT_TMR;
_010: NOP   0;
NETWORK
TITLE = ACCUMULLATOR ON OFF
      A     "ALWAYS_ON";
      A(;
      O     "HYDRAULIC_FUNCTIONS_DB".EMG_ACCM_STA_PB_LCS;
      O     "HYDRAULIC_FUNCTIONS_DB".EMG_ACCM_ON_CMD;
      );
      A     "HYDRAULIC_FUNCTIONS_DB".EMG_ACCM_STP_PB_LCS;
      AN    "HYDRAULIC_FUNCTIONS_DB".PUMP_1_RUN_FB;
      AN    "HYDRAULIC_FUNCTIONS_DB".PUMP_2_RUN_FB;
      =     "HYDRAULIC_FUNCTIONS_DB".EMG_ACCM_ON_CMD;
NETWORK
TITLE = EMERGENCY ACCUMULLATOR ON INDICATOR
      A     "ALWAYS_ON";
      A(;
      O     "HYDRAULIC_FUNCTIONS_DB".EMG_ACCM_ON_CMD;
      O     "HYDRAULIC_FUNCTIONS_DB".LAMP_TEST_PB_LCS_41;
      );
      =     "HYDRAULIC_FUNCTIONS_DB".ACCM_IN_OPER_IND_LCS;
NETWORK
TITLE = COOLER ON INDICATOR
      A     "ALWAYS_ON";
      A(;
      A     "HYDRAULIC_FUNCTIONS_DB".CLR_FAN_ON_CMD;
      A(;
      O     "HALF_SECOND_PULSE_TRAIN";
      O     "HYDRAULIC_FUNCTIONS_DB".COLR_FAN_RUN_FB;
      );
      O     "HYDRAULIC_FUNCTIONS_DB".LAMP_TEST_PB_LCS_41;
      );
      =     "HYDRAULIC_FUNCTIONS_DB".CLR_FAN_ON_IND_LCS;
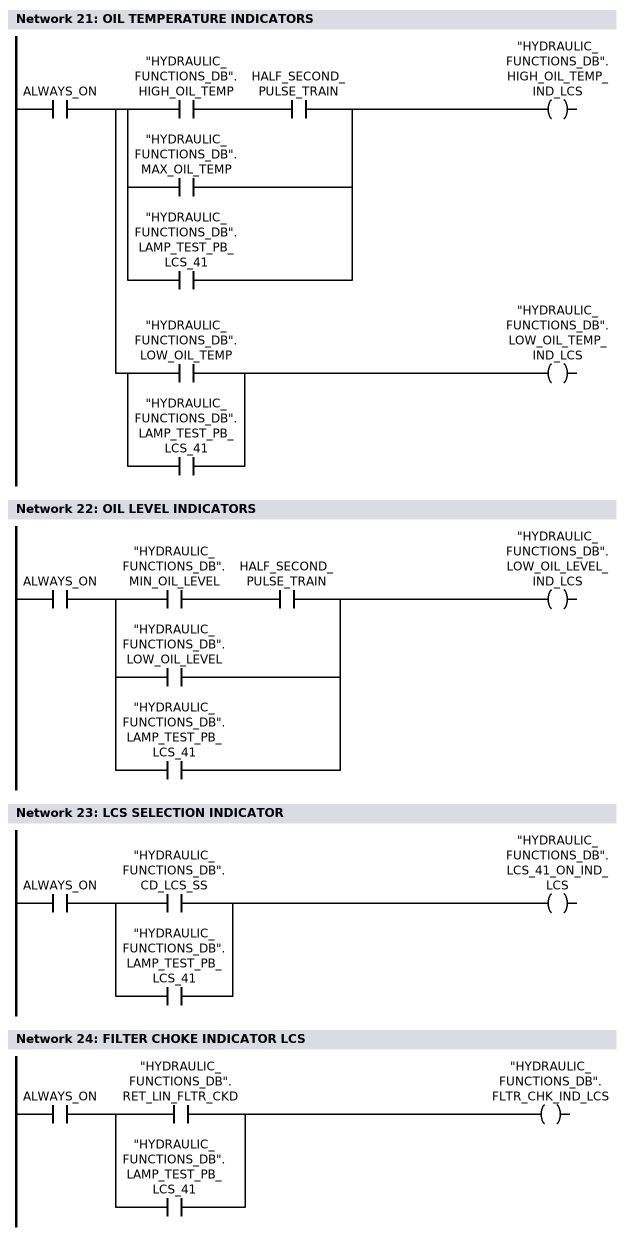
NETWORK
TITLE = OIL TEMPERATURE INDICATORS
      A     "ALWAYS_ON";
      =     L 0.0;
      A     L 0.0;
      A(;
      A     "HYDRAULIC_FUNCTIONS_DB".HIGH_OIL_TEMP;
      A     "HALF_SECOND_PULSE_TRAIN";
      O     "HYDRAULIC_FUNCTIONS_DB".MAX_OIL_TEMP;
      O     "HYDRAULIC_FUNCTIONS_DB".LAMP_TEST_PB_LCS_41;
      );
      =     "HYDRAULIC_FUNCTIONS_DB".HIGH_OIL_TEMP_IND_LCS;
      A     L 0.0;
      A(;
      O     "HYDRAULIC_FUNCTIONS_DB".LOW_OIL_TEMP;
      O     "HYDRAULIC_FUNCTIONS_DB".LAMP_TEST_PB_LCS_41;
      );
      =     "HYDRAULIC_FUNCTIONS_DB".LOW_OIL_TEMP_IND_LCS;
NETWORK
TITLE = OIL LEVEL INDICATORS
      A     "ALWAYS_ON";
      A(;
      A     "HYDRAULIC_FUNCTIONS_DB".MIN_OIL_LEVEL;
      A     "HALF_SECOND_PULSE_TRAIN";
      O     "HYDRAULIC_FUNCTIONS_DB".LOW_OIL_LEVEL;
      O     "HYDRAULIC_FUNCTIONS_DB".LAMP_TEST_PB_LCS_41;
      );
      =     "HYDRAULIC_FUNCTIONS_DB".LOW_OIL_LEVEL_IND_LCS;
NETWORK
TITLE = LCS SELECTION INDICATOR
      A     "ALWAYS_ON";
      A(;
      O     "HYDRAULIC_FUNCTIONS_DB".CD_LCS_SS;
      O     "HYDRAULIC_FUNCTIONS_DB".LAMP_TEST_PB_LCS_41;
      );
      =     "HYDRAULIC_FUNCTIONS_DB".LCS_41_ON_IND_LCS;
NETWORK
TITLE = FILTER CHOKE INDICATOR LCS
      A     "ALWAYS_ON";
      A(;
      O     "HYDRAULIC_FUNCTIONS_DB".RET_LIN_FLTR_CKD;
      O     "HYDRAULIC_FUNCTIONS_DB".LAMP_TEST_PB_LCS_41;
      );
      =     "HYDRAULIC_FUNCTIONS_DB".FLTR_CHK_IND_LCS;
END_FUNCTION

FUNCTION "TRAVEL_DRIVE" : VOID	// FC 5
TITLE = LONG TRAVEL
AUTHOR : Kamillas
VERSION : 0.1
BEGIN
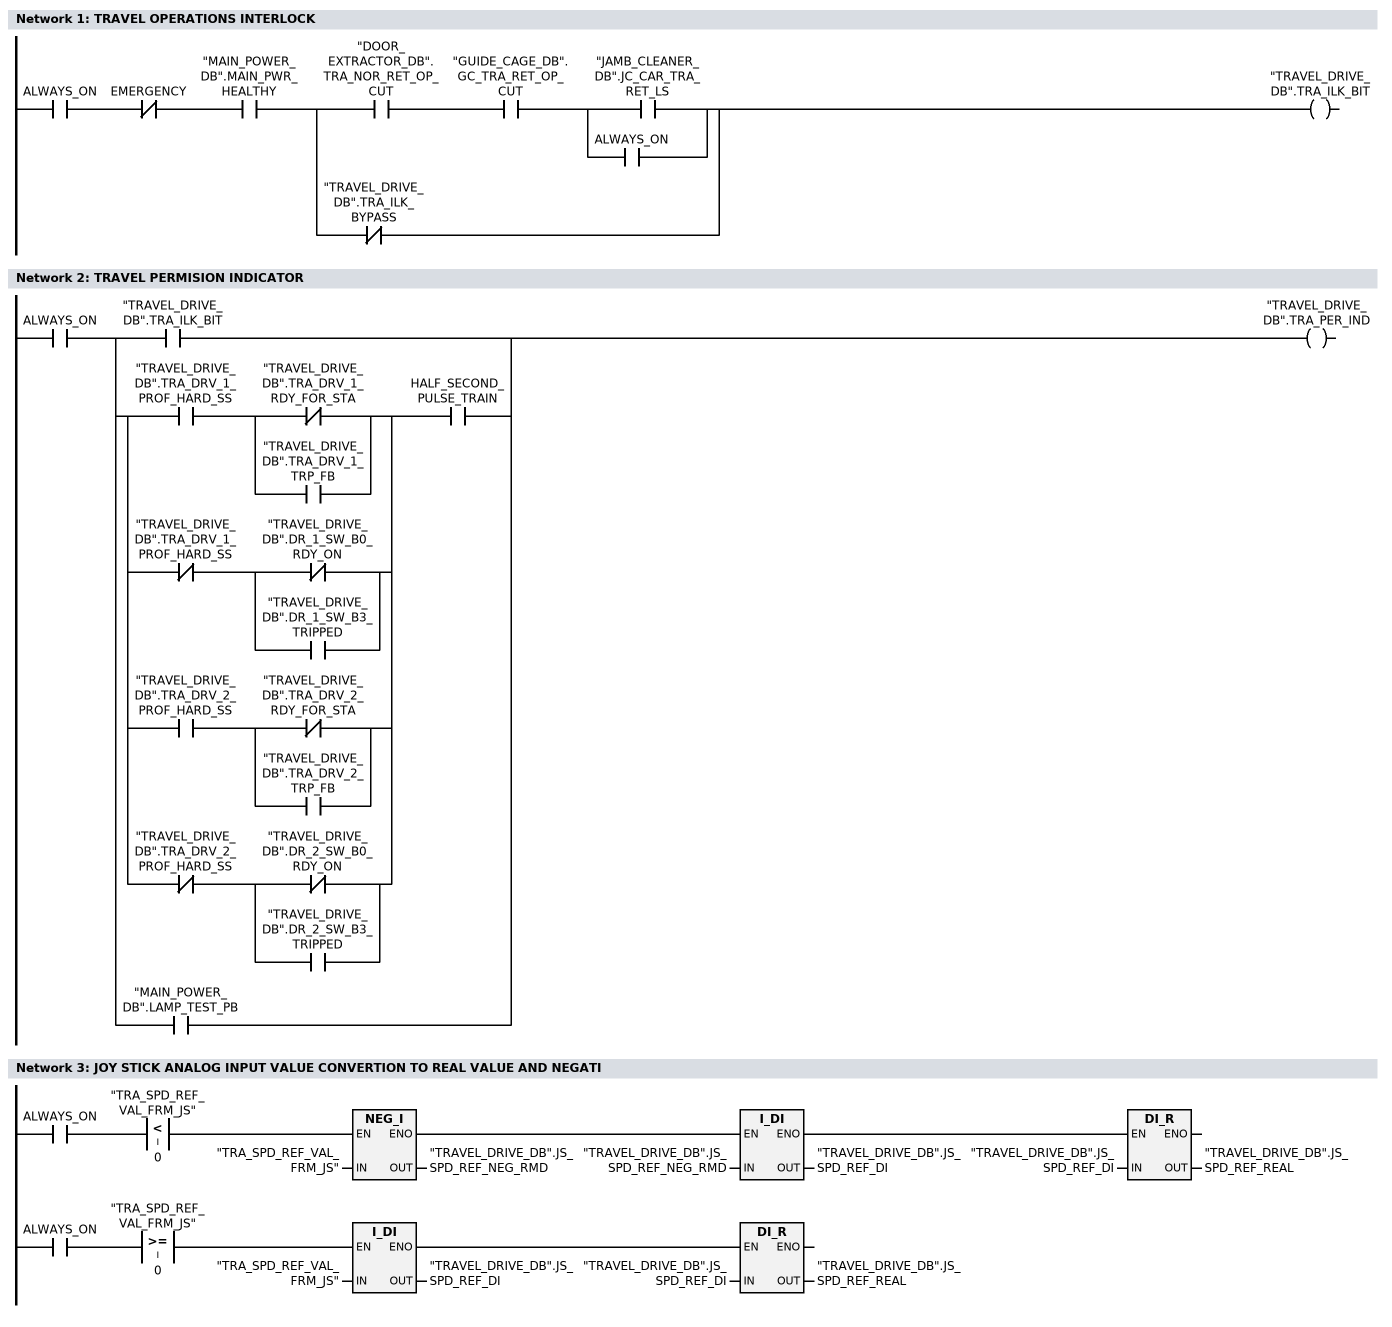
NETWORK
TITLE = TRAVEL OPERATIONS INTERLOCK
      A     "ALWAYS_ON";
      AN    "EMERGENCY";
      A     "MAIN_POWER_DB".MAIN_PWR_HEALTHY;
      A(;
      A     "DOOR_EXTRACTOR_DB".TRA_NOR_RET_OP_CUT;
      A     "GUIDE_CAGE_DB".GC_TRA_RET_OP_CUT;
      A(;
      O     "JAMB_CLEANER_DB".JC_CAR_TRA_RET_LS;
      O     "ALWAYS_ON";
      );
      ON    "TRAVEL_DRIVE_DB".TRA_ILK_BYPASS;
      );
      =     "TRAVEL_DRIVE_DB".TRA_ILK_BIT;
NETWORK
TITLE = TRAVEL PERMISION INDICATOR
      A     "ALWAYS_ON";
      A(;
      O     "TRAVEL_DRIVE_DB".TRA_ILK_BIT;
      O;
      A(;
      A     "TRAVEL_DRIVE_DB".TRA_DRV_1_PROF_HARD_SS;
      A(;
      ON    "TRAVEL_DRIVE_DB".TRA_DRV_1_RDY_FOR_STA;
      O     "TRAVEL_DRIVE_DB".TRA_DRV_1_TRP_FB;
      );
      O;
      AN    "TRAVEL_DRIVE_DB".TRA_DRV_1_PROF_HARD_SS;
      A(;
      ON    "TRAVEL_DRIVE_DB".DR_1_SW_B0_RDY_ON;
      O     "TRAVEL_DRIVE_DB".DR_1_SW_B3_TRIPPED;
      );
      O;
      A     "TRAVEL_DRIVE_DB".TRA_DRV_2_PROF_HARD_SS;
      A(;
      ON    "TRAVEL_DRIVE_DB".TRA_DRV_2_RDY_FOR_STA;
      O     "TRAVEL_DRIVE_DB".TRA_DRV_2_TRP_FB;
      );
      O;
      AN    "TRAVEL_DRIVE_DB".TRA_DRV_2_PROF_HARD_SS;
      A(;
      ON    "TRAVEL_DRIVE_DB".DR_2_SW_B0_RDY_ON;
      O     "TRAVEL_DRIVE_DB".DR_2_SW_B3_TRIPPED;
      );
      );
      A     "HALF_SECOND_PULSE_TRAIN";
      O     "MAIN_POWER_DB".LAMP_TEST_PB;
      );
      =     "TRAVEL_DRIVE_DB".TRA_PER_IND;
NETWORK
TITLE = JOY STICK ANALOG INPUT VALUE CONVERTION TO REAL VALUE AND NEGATI
//JOY STICK ANALOG INPUT VALUE CONVERTION TO REAL VALUE AND NEGATIVE TO POSITIVE 
//CONVERTION
      A     "ALWAYS_ON";
      =     L 0.0;
      A(;
      A(;
      A     L 0.0;
      A(;
      L     "TRA_SPD_REF_VAL_FRM_JS";
      L     0;
      <I;
      );
      JNB   _001;
      L     "TRA_SPD_REF_VAL_FRM_JS";
      NEGI;
      T     "TRAVEL_DRIVE_DB".JS_SPD_REF_NEG_RMD;
      AN    OV;
      SAVE;
      CLR;
_001: A     BR;
      );
      JNB   _002;
      L     "TRAVEL_DRIVE_DB".JS_SPD_REF_NEG_RMD;
      ITD;
      T     "TRAVEL_DRIVE_DB".JS_SPD_REF_DI;
      SET;
      SAVE;
      CLR;
_002: A     BR;
      );
      JNB   _003;
      L     "TRAVEL_DRIVE_DB".JS_SPD_REF_DI;
      DTR;
      T     "TRAVEL_DRIVE_DB".JS_SPD_REF_REAL;
_003: NOP   0;
      A(;
      A     L 0.0;
      A(;
      L     "TRA_SPD_REF_VAL_FRM_JS";
      L     0;
      >=I;
      );
      JNB   _004;
      L     "TRA_SPD_REF_VAL_FRM_JS";
      ITD;
      T     "TRAVEL_DRIVE_DB".JS_SPD_REF_DI;
      SET;
      SAVE;
      CLR;
_004: A     BR;
      );
      JNB   _005;
      L     "TRAVEL_DRIVE_DB".JS_SPD_REF_DI;
      DTR;
      T     "TRAVEL_DRIVE_DB".JS_SPD_REF_REAL;
_005: NOP   0;
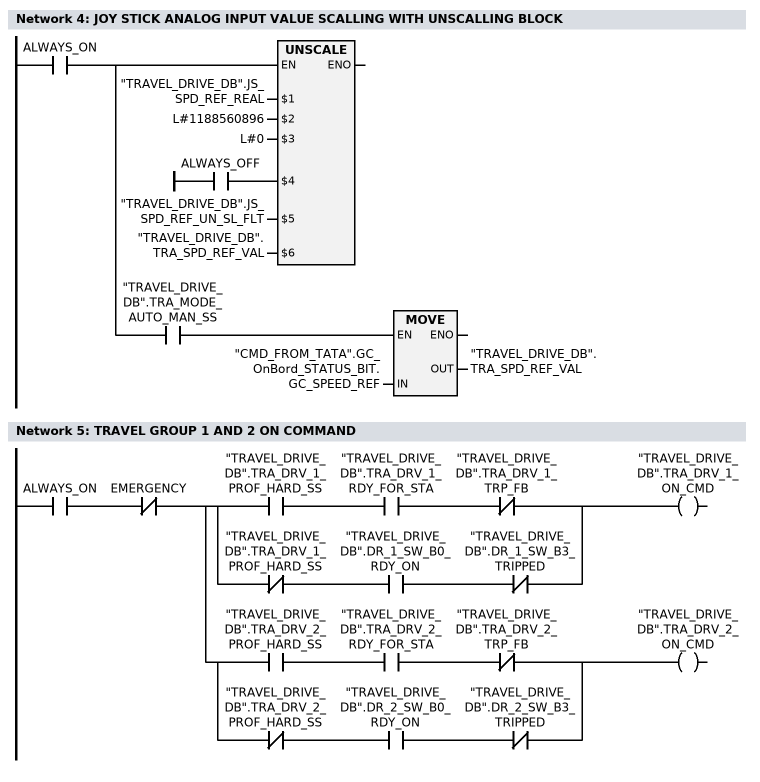
NETWORK
TITLE = JOY STICK ANALOG INPUT VALUE SCALLING WITH UNSCALLING BLOCK
      A     "ALWAYS_ON";
      =     L 0.0;
      A     "ALWAYS_OFF";
      =     L 0.1;
      BLD   103;
      A     L 0.0;
      JNB   _006;
      CALL  "UNSCALE" (
           $1                       := "TRAVEL_DRIVE_DB".JS_SPD_REF_REAL,
           $2                       := L#1188560896,
           $3                       := L#0,
           $4                       := L 0.1,
           $5                       := "TRAVEL_DRIVE_DB".JS_SPD_REF_UN_SL_FLT,
           $6                       := "TRAVEL_DRIVE_DB".TRA_SPD_REF_VAL);
_006: NOP   0;
      A     L 0.0;
      A     "TRAVEL_DRIVE_DB".TRA_MODE_AUTO_MAN_SS;
      JNB   _007;
      L     "CMD_FROM_TATA".GC_OnBord_STATUS_BIT.GC_SPEED_REF;
      T     "TRAVEL_DRIVE_DB".TRA_SPD_REF_VAL;
_007: NOP   0;
NETWORK
TITLE = TRAVEL GROUP 1 AND 2 ON COMMAND
      A     "ALWAYS_ON";
      AN    "EMERGENCY";
      =     L 0.0;
      A     L 0.0;
      A(;
      A     "TRAVEL_DRIVE_DB".TRA_DRV_1_PROF_HARD_SS;
      A     "TRAVEL_DRIVE_DB".TRA_DRV_1_RDY_FOR_STA;
      AN    "TRAVEL_DRIVE_DB".TRA_DRV_1_TRP_FB;
      O;
      AN    "TRAVEL_DRIVE_DB".TRA_DRV_1_PROF_HARD_SS;
      A     "TRAVEL_DRIVE_DB".DR_1_SW_B0_RDY_ON;
      AN    "TRAVEL_DRIVE_DB".DR_1_SW_B3_TRIPPED;
      );
      =     "TRAVEL_DRIVE_DB".TRA_DRV_1_ON_CMD;
      A     L 0.0;
      A(;
      A     "TRAVEL_DRIVE_DB".TRA_DRV_2_PROF_HARD_SS;
      A     "TRAVEL_DRIVE_DB".TRA_DRV_2_RDY_FOR_STA;
      AN    "TRAVEL_DRIVE_DB".TRA_DRV_2_TRP_FB;
      O;
      AN    "TRAVEL_DRIVE_DB".TRA_DRV_2_PROF_HARD_SS;
      A     "TRAVEL_DRIVE_DB".DR_2_SW_B0_RDY_ON;
      AN    "TRAVEL_DRIVE_DB".DR_2_SW_B3_TRIPPED;
      );
      =     "TRAVEL_DRIVE_DB".TRA_DRV_2_ON_CMD;
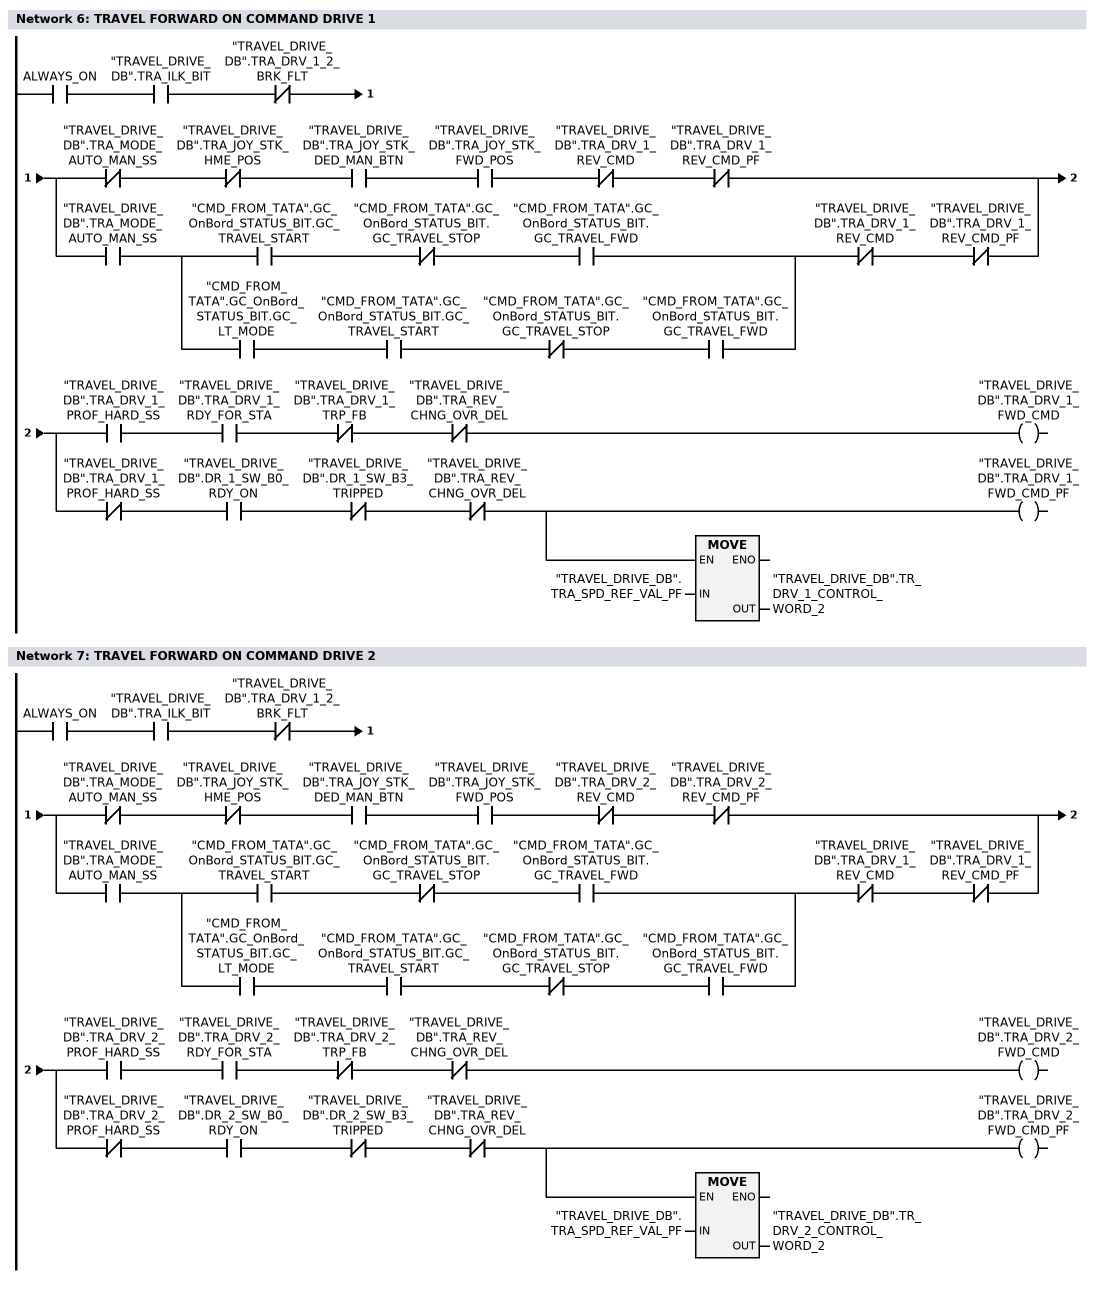
NETWORK
TITLE = TRAVEL FORWARD ON COMMAND DRIVE 1
      A     "ALWAYS_ON";
      A     "TRAVEL_DRIVE_DB".TRA_ILK_BIT;
      AN    "TRAVEL_DRIVE_DB".TRA_DRV_1_2_BRK_FLT;
      A(;
      AN    "TRAVEL_DRIVE_DB".TRA_MODE_AUTO_MAN_SS;
      AN    "TRAVEL_DRIVE_DB".TRA_JOY_STK_HME_POS;
      A     "TRAVEL_DRIVE_DB".TRA_JOY_STK_DED_MAN_BTN;
      A     "TRAVEL_DRIVE_DB".TRA_JOY_STK_FWD_POS;
      AN    "TRAVEL_DRIVE_DB".TRA_DRV_1_REV_CMD;
      AN    "TRAVEL_DRIVE_DB".TRA_DRV_1_REV_CMD_PF;
      O;
      A     "TRAVEL_DRIVE_DB".TRA_MODE_AUTO_MAN_SS;
      A(;
      A     "CMD_FROM_TATA".GC_OnBord_STATUS_BIT.GC_TRAVEL_START;
      AN    "CMD_FROM_TATA".GC_OnBord_STATUS_BIT.GC_TRAVEL_STOP;
      A     "CMD_FROM_TATA".GC_OnBord_STATUS_BIT.GC_TRAVEL_FWD;
      O;
      A     "CMD_FROM_TATA".GC_OnBord_STATUS_BIT.GC_LT_MODE;
      A     "CMD_FROM_TATA".GC_OnBord_STATUS_BIT.GC_TRAVEL_START;
      AN    "CMD_FROM_TATA".GC_OnBord_STATUS_BIT.GC_TRAVEL_STOP;
      A     "CMD_FROM_TATA".GC_OnBord_STATUS_BIT.GC_TRAVEL_FWD;
      );
      AN    "TRAVEL_DRIVE_DB".TRA_DRV_1_REV_CMD;
      AN    "TRAVEL_DRIVE_DB".TRA_DRV_1_REV_CMD_PF;
      );
      =     L 0.0;
      A     L 0.0;
      A     "TRAVEL_DRIVE_DB".TRA_DRV_1_PROF_HARD_SS;
      A     "TRAVEL_DRIVE_DB".TRA_DRV_1_RDY_FOR_STA;
      AN    "TRAVEL_DRIVE_DB".TRA_DRV_1_TRP_FB;
      AN    "TRAVEL_DRIVE_DB".TRA_REV_CHNG_OVR_DEL;
      =     "TRAVEL_DRIVE_DB".TRA_DRV_1_FWD_CMD;
      A     L 0.0;
      AN    "TRAVEL_DRIVE_DB".TRA_DRV_1_PROF_HARD_SS;
      A     "TRAVEL_DRIVE_DB".DR_1_SW_B0_RDY_ON;
      AN    "TRAVEL_DRIVE_DB".DR_1_SW_B3_TRIPPED;
      AN    "TRAVEL_DRIVE_DB".TRA_REV_CHNG_OVR_DEL;
      =     L 0.1;
      A     L 0.1;
      BLD   102;
      =     "TRAVEL_DRIVE_DB".TRA_DRV_1_FWD_CMD_PF;
      A     L 0.1;
      JNB   _008;
      L     "TRAVEL_DRIVE_DB".TRA_SPD_REF_VAL_PF;
      T     "TRAVEL_DRIVE_DB".TR_DRV_1_CONTROL_WORD_2;
_008: NOP   0;
NETWORK
TITLE = TRAVEL FORWARD ON COMMAND DRIVE 2
      A     "ALWAYS_ON";
      A     "TRAVEL_DRIVE_DB".TRA_ILK_BIT;
      AN    "TRAVEL_DRIVE_DB".TRA_DRV_1_2_BRK_FLT;
      A(;
      AN    "TRAVEL_DRIVE_DB".TRA_MODE_AUTO_MAN_SS;
      AN    "TRAVEL_DRIVE_DB".TRA_JOY_STK_HME_POS;
      A     "TRAVEL_DRIVE_DB".TRA_JOY_STK_DED_MAN_BTN;
      A     "TRAVEL_DRIVE_DB".TRA_JOY_STK_FWD_POS;
      AN    "TRAVEL_DRIVE_DB".TRA_DRV_2_REV_CMD;
      AN    "TRAVEL_DRIVE_DB".TRA_DRV_2_REV_CMD_PF;
      O;
      A     "TRAVEL_DRIVE_DB".TRA_MODE_AUTO_MAN_SS;
      A(;
      A     "CMD_FROM_TATA".GC_OnBord_STATUS_BIT.GC_TRAVEL_START;
      AN    "CMD_FROM_TATA".GC_OnBord_STATUS_BIT.GC_TRAVEL_STOP;
      A     "CMD_FROM_TATA".GC_OnBord_STATUS_BIT.GC_TRAVEL_FWD;
      O;
      A     "CMD_FROM_TATA".GC_OnBord_STATUS_BIT.GC_LT_MODE;
      A     "CMD_FROM_TATA".GC_OnBord_STATUS_BIT.GC_TRAVEL_START;
      AN    "CMD_FROM_TATA".GC_OnBord_STATUS_BIT.GC_TRAVEL_STOP;
      A     "CMD_FROM_TATA".GC_OnBord_STATUS_BIT.GC_TRAVEL_FWD;
      );
      AN    "TRAVEL_DRIVE_DB".TRA_DRV_1_REV_CMD;
      AN    "TRAVEL_DRIVE_DB".TRA_DRV_1_REV_CMD_PF;
      );
      =     L 0.0;
      A     L 0.0;
      A     "TRAVEL_DRIVE_DB".TRA_DRV_2_PROF_HARD_SS;
      A     "TRAVEL_DRIVE_DB".TRA_DRV_2_RDY_FOR_STA;
      AN    "TRAVEL_DRIVE_DB".TRA_DRV_2_TRP_FB;
      AN    "TRAVEL_DRIVE_DB".TRA_REV_CHNG_OVR_DEL;
      =     "TRAVEL_DRIVE_DB".TRA_DRV_2_FWD_CMD;
      A     L 0.0;
      AN    "TRAVEL_DRIVE_DB".TRA_DRV_2_PROF_HARD_SS;
      A     "TRAVEL_DRIVE_DB".DR_2_SW_B0_RDY_ON;
      AN    "TRAVEL_DRIVE_DB".DR_2_SW_B3_TRIPPED;
      AN    "TRAVEL_DRIVE_DB".TRA_REV_CHNG_OVR_DEL;
      =     L 0.1;
      A     L 0.1;
      BLD   102;
      =     "TRAVEL_DRIVE_DB".TRA_DRV_2_FWD_CMD_PF;
      A     L 0.1;
      JNB   _009;
      L     "TRAVEL_DRIVE_DB".TRA_SPD_REF_VAL_PF;
      T     "TRAVEL_DRIVE_DB".TR_DRV_2_CONTROL_WORD_2;
_009: NOP   0;
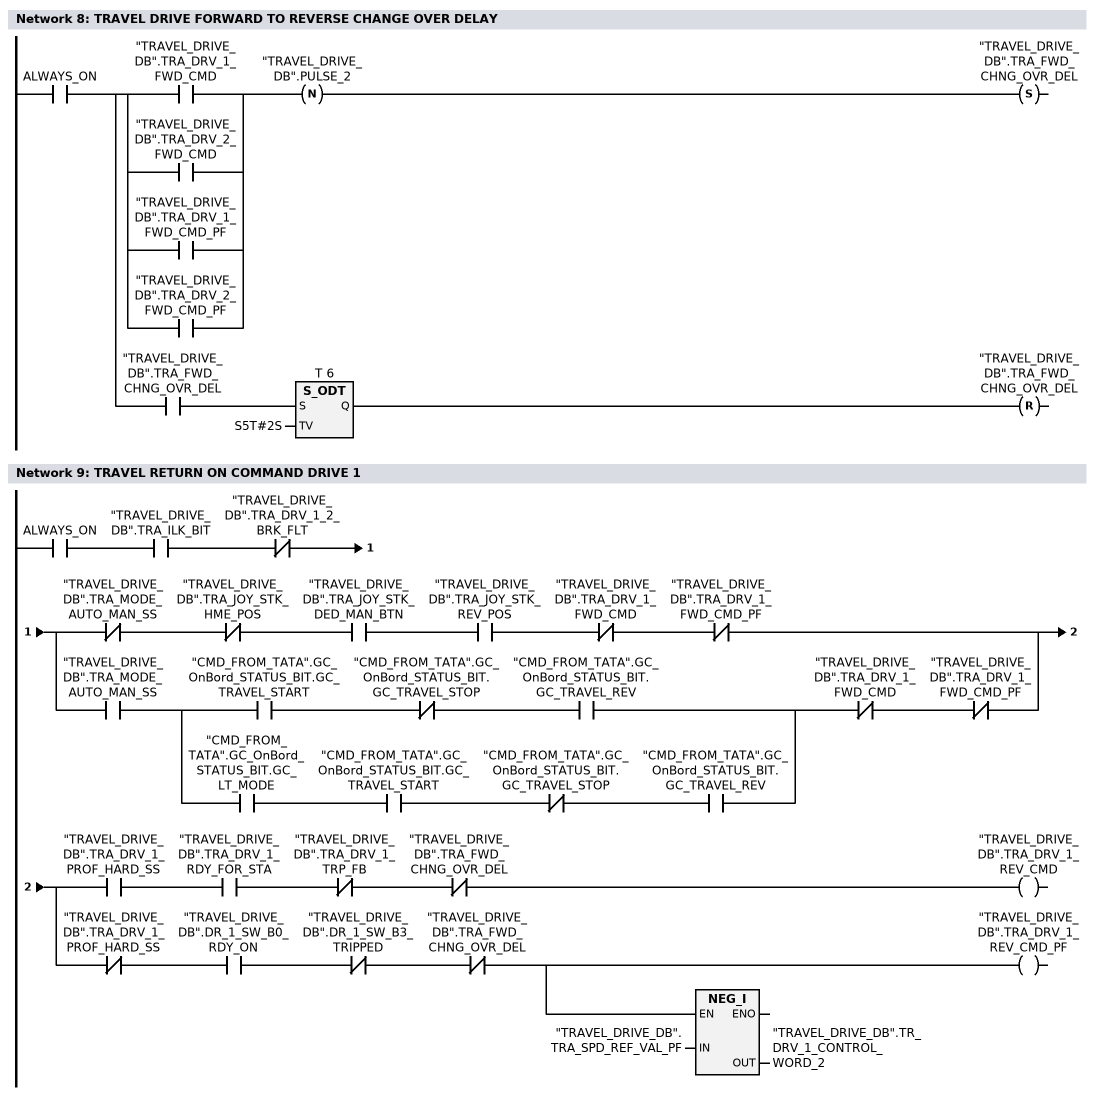
NETWORK
TITLE = TRAVEL DRIVE FORWARD TO REVERSE CHANGE OVER DELAY
      A     "ALWAYS_ON";
      =     L 0.0;
      A     L 0.0;
      A(;
      O     "TRAVEL_DRIVE_DB".TRA_DRV_1_FWD_CMD;
      O     "TRAVEL_DRIVE_DB".TRA_DRV_2_FWD_CMD;
      O     "TRAVEL_DRIVE_DB".TRA_DRV_1_FWD_CMD_PF;
      O     "TRAVEL_DRIVE_DB".TRA_DRV_2_FWD_CMD_PF;
      );
      FN    "TRAVEL_DRIVE_DB".PULSE_2;
      S     "TRAVEL_DRIVE_DB".TRA_FWD_CHNG_OVR_DEL;
      A     L 0.0;
      A     "TRAVEL_DRIVE_DB".TRA_FWD_CHNG_OVR_DEL;
      L     S5T#2S;
      SD    T 6;
      NOP   0;
      NOP   0;
      NOP   0;
      A     T 6;
      R     "TRAVEL_DRIVE_DB".TRA_FWD_CHNG_OVR_DEL;
NETWORK
TITLE = TRAVEL RETURN ON COMMAND DRIVE 1
      A     "ALWAYS_ON";
      A     "TRAVEL_DRIVE_DB".TRA_ILK_BIT;
      AN    "TRAVEL_DRIVE_DB".TRA_DRV_1_2_BRK_FLT;
      A(;
      AN    "TRAVEL_DRIVE_DB".TRA_MODE_AUTO_MAN_SS;
      AN    "TRAVEL_DRIVE_DB".TRA_JOY_STK_HME_POS;
      A     "TRAVEL_DRIVE_DB".TRA_JOY_STK_DED_MAN_BTN;
      A     "TRAVEL_DRIVE_DB".TRA_JOY_STK_REV_POS;
      AN    "TRAVEL_DRIVE_DB".TRA_DRV_1_FWD_CMD;
      AN    "TRAVEL_DRIVE_DB".TRA_DRV_1_FWD_CMD_PF;
      O;
      A     "TRAVEL_DRIVE_DB".TRA_MODE_AUTO_MAN_SS;
      A(;
      A     "CMD_FROM_TATA".GC_OnBord_STATUS_BIT.GC_TRAVEL_START;
      AN    "CMD_FROM_TATA".GC_OnBord_STATUS_BIT.GC_TRAVEL_STOP;
      A     "CMD_FROM_TATA".GC_OnBord_STATUS_BIT.GC_TRAVEL_REV;
      O;
      A     "CMD_FROM_TATA".GC_OnBord_STATUS_BIT.GC_LT_MODE;
      A     "CMD_FROM_TATA".GC_OnBord_STATUS_BIT.GC_TRAVEL_START;
      AN    "CMD_FROM_TATA".GC_OnBord_STATUS_BIT.GC_TRAVEL_STOP;
      A     "CMD_FROM_TATA".GC_OnBord_STATUS_BIT.GC_TRAVEL_REV;
      );
      AN    "TRAVEL_DRIVE_DB".TRA_DRV_1_FWD_CMD;
      AN    "TRAVEL_DRIVE_DB".TRA_DRV_1_FWD_CMD_PF;
      );
      =     L 0.0;
      A     L 0.0;
      A     "TRAVEL_DRIVE_DB".TRA_DRV_1_PROF_HARD_SS;
      A     "TRAVEL_DRIVE_DB".TRA_DRV_1_RDY_FOR_STA;
      AN    "TRAVEL_DRIVE_DB".TRA_DRV_1_TRP_FB;
      AN    "TRAVEL_DRIVE_DB".TRA_FWD_CHNG_OVR_DEL;
      =     "TRAVEL_DRIVE_DB".TRA_DRV_1_REV_CMD;
      A     L 0.0;
      AN    "TRAVEL_DRIVE_DB".TRA_DRV_1_PROF_HARD_SS;
      A     "TRAVEL_DRIVE_DB".DR_1_SW_B0_RDY_ON;
      AN    "TRAVEL_DRIVE_DB".DR_1_SW_B3_TRIPPED;
      AN    "TRAVEL_DRIVE_DB".TRA_FWD_CHNG_OVR_DEL;
      =     L 0.1;
      A     L 0.1;
      BLD   102;
      =     "TRAVEL_DRIVE_DB".TRA_DRV_1_REV_CMD_PF;
      A     L 0.1;
      JNB   _00a;
      L     "TRAVEL_DRIVE_DB".TRA_SPD_REF_VAL_PF;
      NEGI;
      T     "TRAVEL_DRIVE_DB".TR_DRV_1_CONTROL_WORD_2;
_00a: NOP   0;
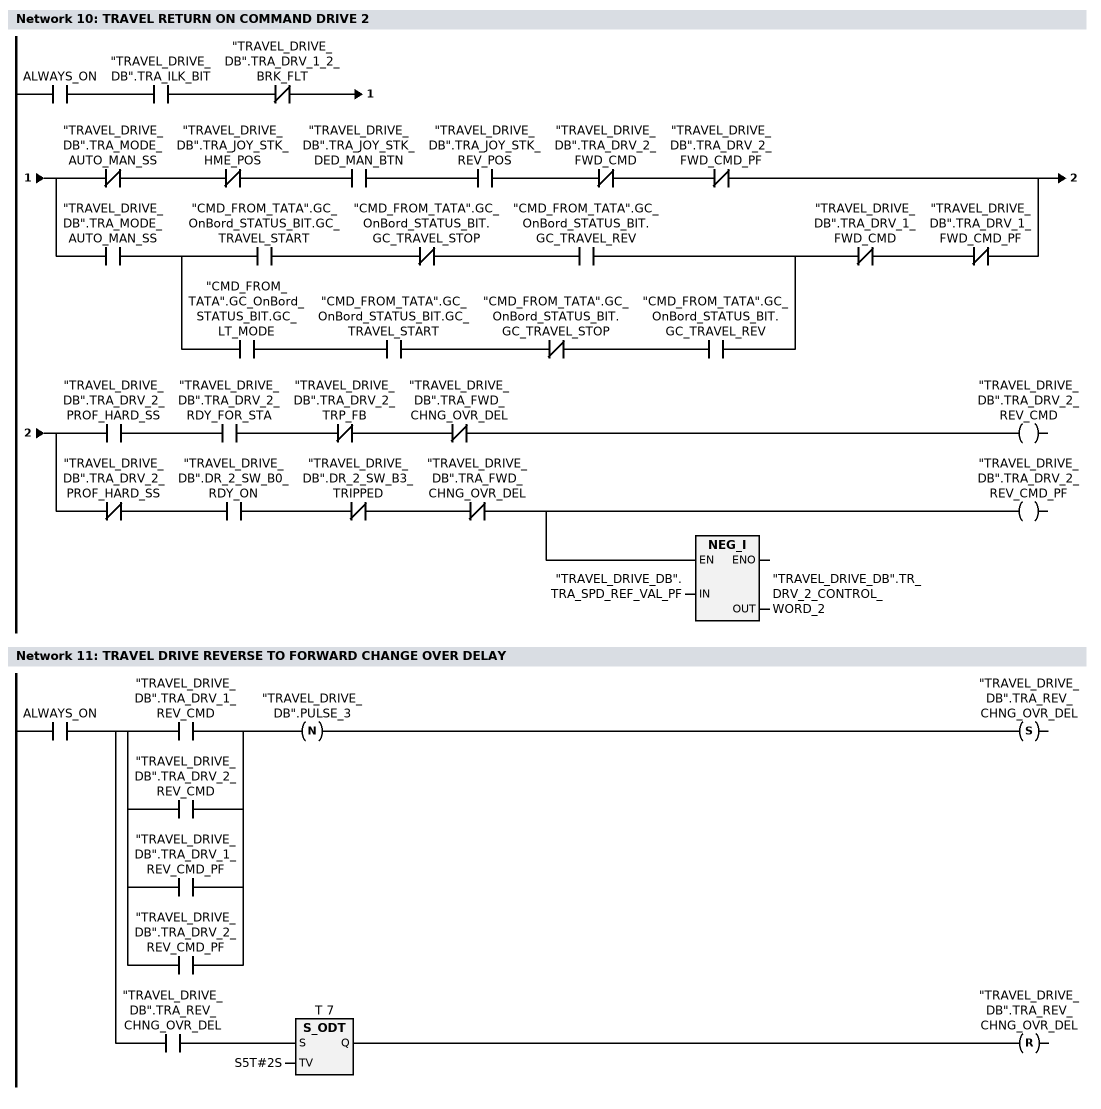
NETWORK
TITLE = TRAVEL RETURN ON COMMAND DRIVE 2
      A     "ALWAYS_ON";
      A     "TRAVEL_DRIVE_DB".TRA_ILK_BIT;
      AN    "TRAVEL_DRIVE_DB".TRA_DRV_1_2_BRK_FLT;
      A(;
      AN    "TRAVEL_DRIVE_DB".TRA_MODE_AUTO_MAN_SS;
      AN    "TRAVEL_DRIVE_DB".TRA_JOY_STK_HME_POS;
      A     "TRAVEL_DRIVE_DB".TRA_JOY_STK_DED_MAN_BTN;
      A     "TRAVEL_DRIVE_DB".TRA_JOY_STK_REV_POS;
      AN    "TRAVEL_DRIVE_DB".TRA_DRV_2_FWD_CMD;
      AN    "TRAVEL_DRIVE_DB".TRA_DRV_2_FWD_CMD_PF;
      O;
      A     "TRAVEL_DRIVE_DB".TRA_MODE_AUTO_MAN_SS;
      A(;
      A     "CMD_FROM_TATA".GC_OnBord_STATUS_BIT.GC_TRAVEL_START;
      AN    "CMD_FROM_TATA".GC_OnBord_STATUS_BIT.GC_TRAVEL_STOP;
      A     "CMD_FROM_TATA".GC_OnBord_STATUS_BIT.GC_TRAVEL_REV;
      O;
      A     "CMD_FROM_TATA".GC_OnBord_STATUS_BIT.GC_LT_MODE;
      A     "CMD_FROM_TATA".GC_OnBord_STATUS_BIT.GC_TRAVEL_START;
      AN    "CMD_FROM_TATA".GC_OnBord_STATUS_BIT.GC_TRAVEL_STOP;
      A     "CMD_FROM_TATA".GC_OnBord_STATUS_BIT.GC_TRAVEL_REV;
      );
      AN    "TRAVEL_DRIVE_DB".TRA_DRV_1_FWD_CMD;
      AN    "TRAVEL_DRIVE_DB".TRA_DRV_1_FWD_CMD_PF;
      );
      =     L 0.0;
      A     L 0.0;
      A     "TRAVEL_DRIVE_DB".TRA_DRV_2_PROF_HARD_SS;
      A     "TRAVEL_DRIVE_DB".TRA_DRV_2_RDY_FOR_STA;
      AN    "TRAVEL_DRIVE_DB".TRA_DRV_2_TRP_FB;
      AN    "TRAVEL_DRIVE_DB".TRA_FWD_CHNG_OVR_DEL;
      =     "TRAVEL_DRIVE_DB".TRA_DRV_2_REV_CMD;
      A     L 0.0;
      AN    "TRAVEL_DRIVE_DB".TRA_DRV_2_PROF_HARD_SS;
      A     "TRAVEL_DRIVE_DB".DR_2_SW_B0_RDY_ON;
      AN    "TRAVEL_DRIVE_DB".DR_2_SW_B3_TRIPPED;
      AN    "TRAVEL_DRIVE_DB".TRA_FWD_CHNG_OVR_DEL;
      =     L 0.1;
      A     L 0.1;
      BLD   102;
      =     "TRAVEL_DRIVE_DB".TRA_DRV_2_REV_CMD_PF;
      A     L 0.1;
      JNB   _00b;
      L     "TRAVEL_DRIVE_DB".TRA_SPD_REF_VAL_PF;
      NEGI;
      T     "TRAVEL_DRIVE_DB".TR_DRV_2_CONTROL_WORD_2;
_00b: NOP   0;
NETWORK
TITLE = TRAVEL DRIVE REVERSE TO FORWARD CHANGE OVER DELAY
      A     "ALWAYS_ON";
      =     L 0.0;
      A     L 0.0;
      A(;
      O     "TRAVEL_DRIVE_DB".TRA_DRV_1_REV_CMD;
      O     "TRAVEL_DRIVE_DB".TRA_DRV_2_REV_CMD;
      O     "TRAVEL_DRIVE_DB".TRA_DRV_1_REV_CMD_PF;
      O     "TRAVEL_DRIVE_DB".TRA_DRV_2_REV_CMD_PF;
      );
      FN    "TRAVEL_DRIVE_DB".PULSE_3;
      S     "TRAVEL_DRIVE_DB".TRA_REV_CHNG_OVR_DEL;
      A     L 0.0;
      A     "TRAVEL_DRIVE_DB".TRA_REV_CHNG_OVR_DEL;
      L     S5T#2S;
      SD    T 7;
      NOP   0;
      NOP   0;
      NOP   0;
      A     T 7;
      R     "TRAVEL_DRIVE_DB".TRA_REV_CHNG_OVR_DEL;
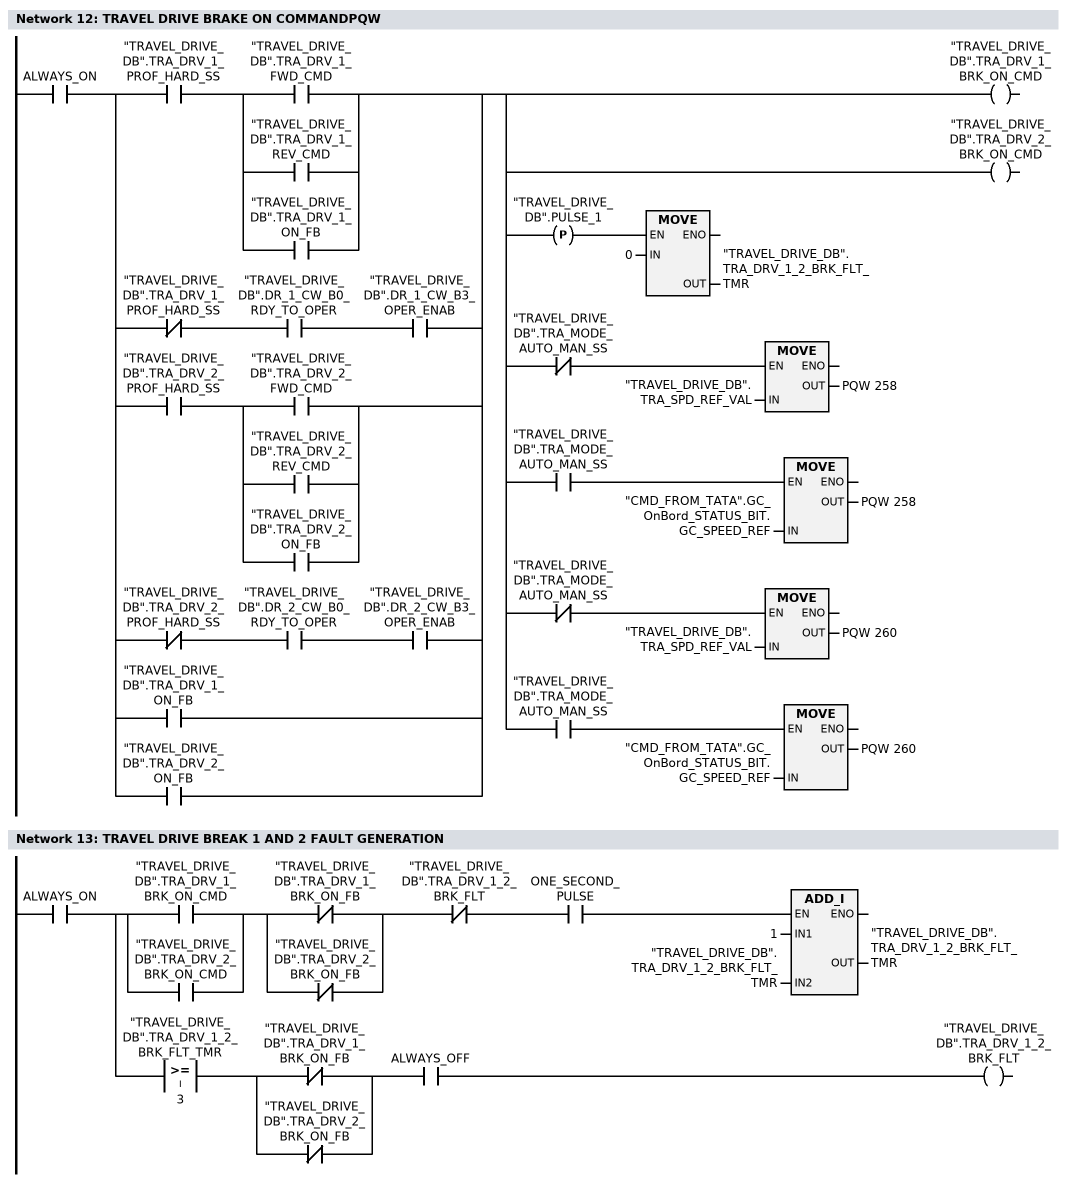
NETWORK
TITLE = TRAVEL DRIVE BRAKE ON COMMANDPQW
      A     "ALWAYS_ON";
      A(;
      A     "TRAVEL_DRIVE_DB".TRA_DRV_1_PROF_HARD_SS;
      A(;
      O     "TRAVEL_DRIVE_DB".TRA_DRV_1_FWD_CMD;
      O     "TRAVEL_DRIVE_DB".TRA_DRV_1_REV_CMD;
      O     "TRAVEL_DRIVE_DB".TRA_DRV_1_ON_FB;
      );
      O;
      AN    "TRAVEL_DRIVE_DB".TRA_DRV_1_PROF_HARD_SS;
      A     "TRAVEL_DRIVE_DB".DR_1_CW_B0_RDY_TO_OPER;
      A     "TRAVEL_DRIVE_DB".DR_1_CW_B3_OPER_ENAB;
      O;
      A     "TRAVEL_DRIVE_DB".TRA_DRV_2_PROF_HARD_SS;
      A(;
      O     "TRAVEL_DRIVE_DB".TRA_DRV_2_FWD_CMD;
      O     "TRAVEL_DRIVE_DB".TRA_DRV_2_REV_CMD;
      O     "TRAVEL_DRIVE_DB".TRA_DRV_2_ON_FB;
      );
      O;
      AN    "TRAVEL_DRIVE_DB".TRA_DRV_2_PROF_HARD_SS;
      A     "TRAVEL_DRIVE_DB".DR_2_CW_B0_RDY_TO_OPER;
      A     "TRAVEL_DRIVE_DB".DR_2_CW_B3_OPER_ENAB;
      O     "TRAVEL_DRIVE_DB".TRA_DRV_1_ON_FB;
      O     "TRAVEL_DRIVE_DB".TRA_DRV_2_ON_FB;
      );
      =     L 0.0;
      A     L 0.0;
      BLD   102;
      =     "TRAVEL_DRIVE_DB".TRA_DRV_1_BRK_ON_CMD;
      A     L 0.0;
      BLD   102;
      =     "TRAVEL_DRIVE_DB".TRA_DRV_2_BRK_ON_CMD;
      A     L 0.0;
      FP    "TRAVEL_DRIVE_DB".PULSE_1;
      JNB   _00c;
      L     0;
      T     "TRAVEL_DRIVE_DB".TRA_DRV_1_2_BRK_FLT_TMR;
_00c: NOP   0;
      A     L 0.0;
      AN    "TRAVEL_DRIVE_DB".TRA_MODE_AUTO_MAN_SS;
      JNB   _00d;
      L     "TRAVEL_DRIVE_DB".TRA_SPD_REF_VAL;
      T     PQW 258;
_00d: NOP   0;
      A     L 0.0;
      A     "TRAVEL_DRIVE_DB".TRA_MODE_AUTO_MAN_SS;
      JNB   _00e;
      L     "CMD_FROM_TATA".GC_OnBord_STATUS_BIT.GC_SPEED_REF;
      T     PQW 258;
_00e: NOP   0;
      A     L 0.0;
      AN    "TRAVEL_DRIVE_DB".TRA_MODE_AUTO_MAN_SS;
      JNB   _00f;
      L     "TRAVEL_DRIVE_DB".TRA_SPD_REF_VAL;
      T     PQW 260;
_00f: NOP   0;
      A     L 0.0;
      A     "TRAVEL_DRIVE_DB".TRA_MODE_AUTO_MAN_SS;
      JNB   _010;
      L     "CMD_FROM_TATA".GC_OnBord_STATUS_BIT.GC_SPEED_REF;
      T     PQW 260;
_010: NOP   0;
NETWORK
TITLE = TRAVEL DRIVE BREAK 1 AND 2 FAULT GENERATION
      A     "ALWAYS_ON";
      =     L 0.0;
      A     L 0.0;
      A(;
      O     "TRAVEL_DRIVE_DB".TRA_DRV_1_BRK_ON_CMD;
      O     "TRAVEL_DRIVE_DB".TRA_DRV_2_BRK_ON_CMD;
      );
      A(;
      ON    "TRAVEL_DRIVE_DB".TRA_DRV_1_BRK_ON_FB;
      ON    "TRAVEL_DRIVE_DB".TRA_DRV_2_BRK_ON_FB;
      );
      AN    "TRAVEL_DRIVE_DB".TRA_DRV_1_2_BRK_FLT;
      A     "ONE_SECOND_PULSE";
      JNB   _011;
      L     1;
      L     "TRAVEL_DRIVE_DB".TRA_DRV_1_2_BRK_FLT_TMR;
      +I;
      T     "TRAVEL_DRIVE_DB".TRA_DRV_1_2_BRK_FLT_TMR;
_011: NOP   0;
      A     L 0.0;
      A(;
      L     "TRAVEL_DRIVE_DB".TRA_DRV_1_2_BRK_FLT_TMR;
      L     3;
      >=I;
      );
      A(;
      ON    "TRAVEL_DRIVE_DB".TRA_DRV_1_BRK_ON_FB;
      ON    "TRAVEL_DRIVE_DB".TRA_DRV_2_BRK_ON_FB;
      );
      A     "ALWAYS_OFF";
      =     "TRAVEL_DRIVE_DB".TRA_DRV_1_2_BRK_FLT;
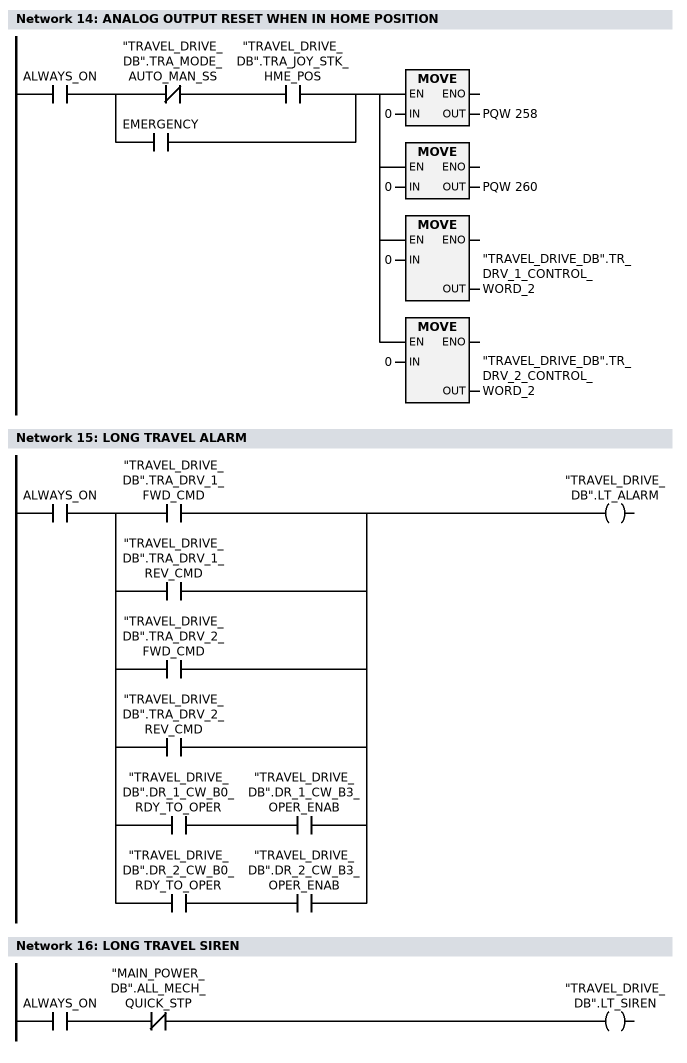
NETWORK
TITLE = ANALOG OUTPUT RESET WHEN IN HOME POSITION
      A     "ALWAYS_ON";
      A(;
      AN    "TRAVEL_DRIVE_DB".TRA_MODE_AUTO_MAN_SS;
      A     "TRAVEL_DRIVE_DB".TRA_JOY_STK_HME_POS;
      O     "EMERGENCY";
      );
      =     L 0.0;
      A     L 0.0;
      JNB   _012;
      L     0;
      T     PQW 258;
_012: NOP   0;
      A     L 0.0;
      JNB   _013;
      L     0;
      T     PQW 260;
_013: NOP   0;
      A     L 0.0;
      JNB   _014;
      L     0;
      T     "TRAVEL_DRIVE_DB".TR_DRV_1_CONTROL_WORD_2;
_014: NOP   0;
      A     L 0.0;
      JNB   _015;
      L     0;
      T     "TRAVEL_DRIVE_DB".TR_DRV_2_CONTROL_WORD_2;
_015: NOP   0;
NETWORK
TITLE = LONG TRAVEL ALARM
      A     "ALWAYS_ON";
      A(;
      O     "TRAVEL_DRIVE_DB".TRA_DRV_1_FWD_CMD;
      O     "TRAVEL_DRIVE_DB".TRA_DRV_1_REV_CMD;
      O     "TRAVEL_DRIVE_DB".TRA_DRV_2_FWD_CMD;
      O     "TRAVEL_DRIVE_DB".TRA_DRV_2_REV_CMD;
      O;
      A     "TRAVEL_DRIVE_DB".DR_1_CW_B0_RDY_TO_OPER;
      A     "TRAVEL_DRIVE_DB".DR_1_CW_B3_OPER_ENAB;
      O;
      A     "TRAVEL_DRIVE_DB".DR_2_CW_B0_RDY_TO_OPER;
      A     "TRAVEL_DRIVE_DB".DR_2_CW_B3_OPER_ENAB;
      );
      =     "TRAVEL_DRIVE_DB".LT_ALARM;
NETWORK
TITLE = LONG TRAVEL SIREN
      A     "ALWAYS_ON";
      AN    "MAIN_POWER_DB".ALL_MECH_QUICK_STP;
      =     "TRAVEL_DRIVE_DB".LT_SIREN;
END_FUNCTION

FUNCTION "AIR_COMPRESSOR" : VOID	// FC 6
TITLE = AIR COMPRESSOR SYSTEM
AUTHOR : Kamillas
VERSION : 0.1
BEGIN
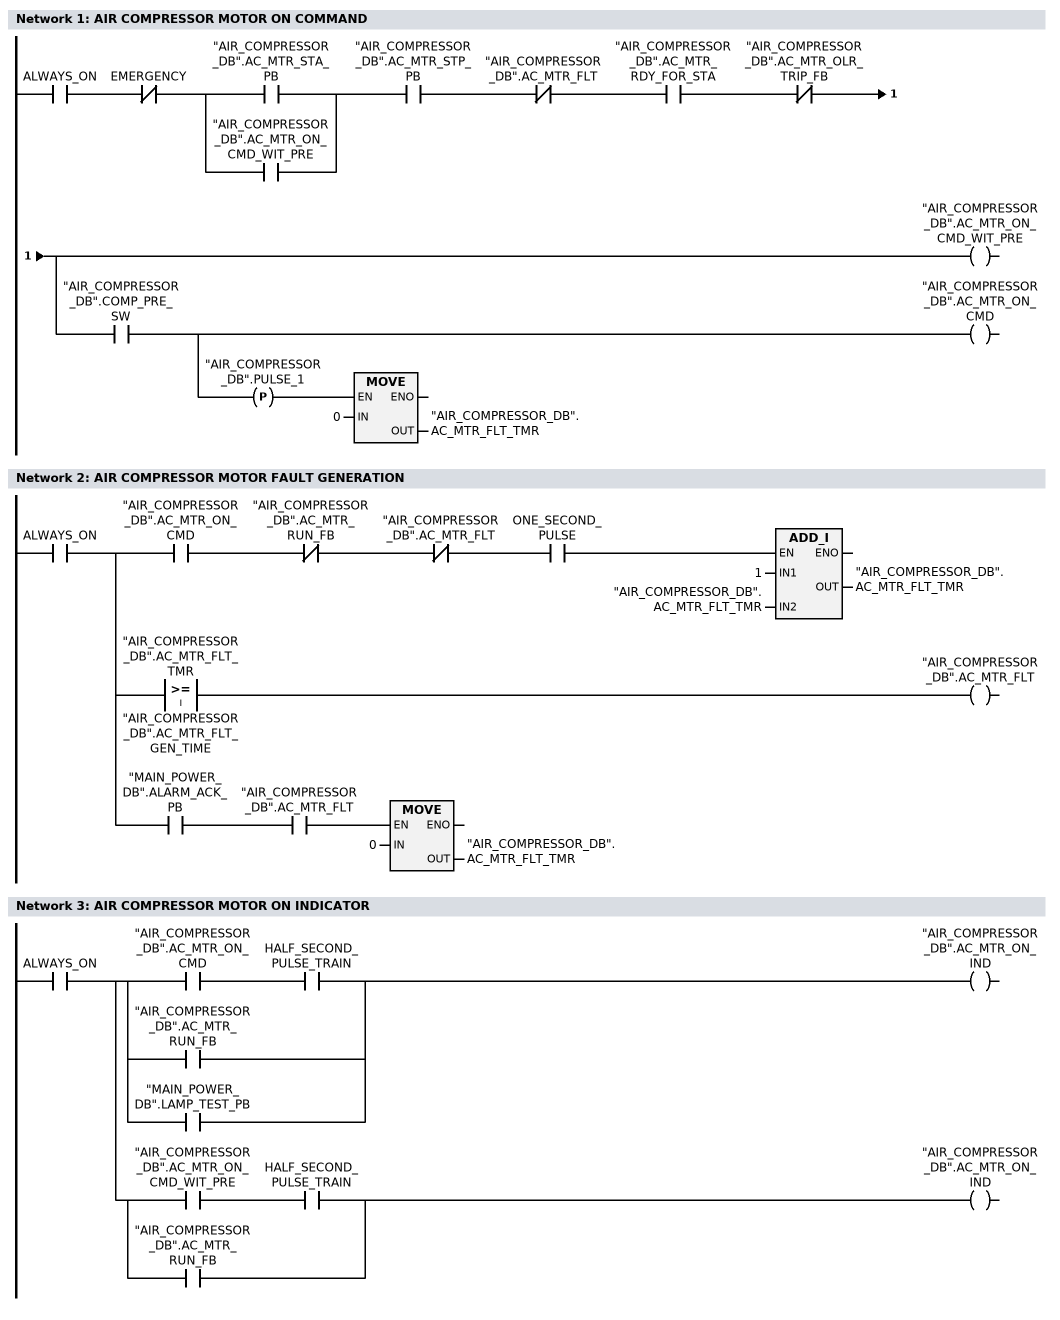
NETWORK
TITLE = AIR COMPRESSOR MOTOR ON COMMAND
      A     "ALWAYS_ON";
      AN    "EMERGENCY";
      A(;
      O     "AIR_COMPRESSOR_DB".AC_MTR_STA_PB;
      O     "AIR_COMPRESSOR_DB".AC_MTR_ON_CMD_WIT_PRE;
      );
      A     "AIR_COMPRESSOR_DB".AC_MTR_STP_PB;
      AN    "AIR_COMPRESSOR_DB".AC_MTR_FLT;
      A     "AIR_COMPRESSOR_DB".AC_MTR_RDY_FOR_STA;
      AN    "AIR_COMPRESSOR_DB".AC_MTR_OLR_TRIP_FB;
      =     L 0.0;
      A     L 0.0;
      BLD   102;
      =     "AIR_COMPRESSOR_DB".AC_MTR_ON_CMD_WIT_PRE;
      A     L 0.0;
      A     "AIR_COMPRESSOR_DB".COMP_PRE_SW;
      =     L 0.1;
      A     L 0.1;
      BLD   102;
      =     "AIR_COMPRESSOR_DB".AC_MTR_ON_CMD;
      A     L 0.1;
      FP    "AIR_COMPRESSOR_DB".PULSE_1;
      JNB   _001;
      L     0;
      T     "AIR_COMPRESSOR_DB".AC_MTR_FLT_TMR;
_001: NOP   0;
NETWORK
TITLE = AIR COMPRESSOR MOTOR FAULT GENERATION
      A     "ALWAYS_ON";
      =     L 0.0;
      A     L 0.0;
      A     "AIR_COMPRESSOR_DB".AC_MTR_ON_CMD;
      AN    "AIR_COMPRESSOR_DB".AC_MTR_RUN_FB;
      AN    "AIR_COMPRESSOR_DB".AC_MTR_FLT;
      A     "ONE_SECOND_PULSE";
      JNB   _002;
      L     1;
      L     "AIR_COMPRESSOR_DB".AC_MTR_FLT_TMR;
      +I;
      T     "AIR_COMPRESSOR_DB".AC_MTR_FLT_TMR;
_002: NOP   0;
      A     L 0.0;
      A(;
      L     "AIR_COMPRESSOR_DB".AC_MTR_FLT_TMR;
      L     "AIR_COMPRESSOR_DB".AC_MTR_FLT_GEN_TIME;
      >=I;
      );
      =     "AIR_COMPRESSOR_DB".AC_MTR_FLT;
      A     L 0.0;
      A     "MAIN_POWER_DB".ALARM_ACK_PB;
      A     "AIR_COMPRESSOR_DB".AC_MTR_FLT;
      JNB   _003;
      L     0;
      T     "AIR_COMPRESSOR_DB".AC_MTR_FLT_TMR;
_003: NOP   0;
NETWORK
TITLE = AIR COMPRESSOR MOTOR ON INDICATOR
      A     "ALWAYS_ON";
      =     L 0.0;
      A     L 0.0;
      A(;
      A     "AIR_COMPRESSOR_DB".AC_MTR_ON_CMD;
      A     "HALF_SECOND_PULSE_TRAIN";
      O     "AIR_COMPRESSOR_DB".AC_MTR_RUN_FB;
      O     "MAIN_POWER_DB".LAMP_TEST_PB;
      );
      =     "AIR_COMPRESSOR_DB".AC_MTR_ON_IND;
      A     L 0.0;
      A(;
      A     "AIR_COMPRESSOR_DB".AC_MTR_ON_CMD_WIT_PRE;
      A     "HALF_SECOND_PULSE_TRAIN";
      O     "AIR_COMPRESSOR_DB".AC_MTR_RUN_FB;
      );
      =     "AIR_COMPRESSOR_DB".AC_MTR_ON_IND;
END_FUNCTION

FUNCTION "HOOD_SYSTEM" : VOID	// FC 7
AUTHOR : Kamillas
VERSION : 0.1
BEGIN
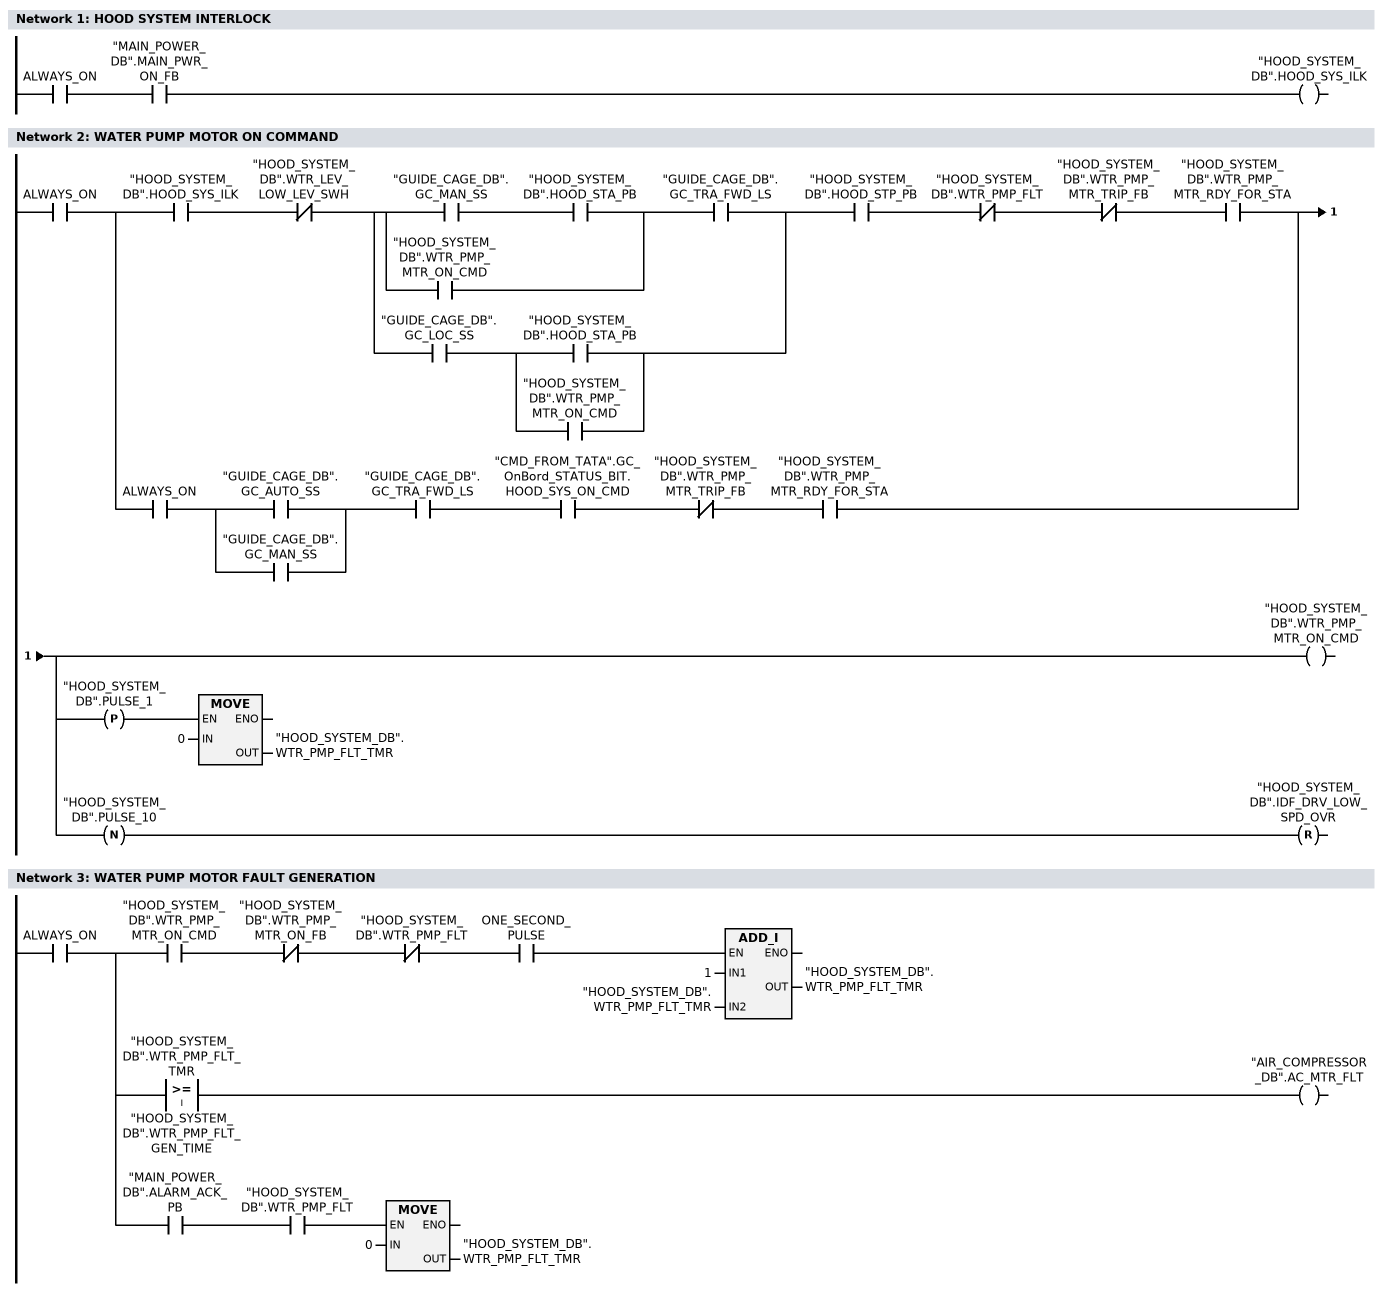
NETWORK
TITLE = HOOD SYSTEM INTERLOCK
      A     "ALWAYS_ON";
      A     "MAIN_POWER_DB".MAIN_PWR_ON_FB;
      =     "HOOD_SYSTEM_DB".HOOD_SYS_ILK;
NETWORK
TITLE = WATER PUMP MOTOR ON COMMAND
      A     "ALWAYS_ON";
      A(;
      A     "HOOD_SYSTEM_DB".HOOD_SYS_ILK;
      AN    "HOOD_SYSTEM_DB".WTR_LEV_LOW_LEV_SWH;
      A(;
      A(;
      A     "GUIDE_CAGE_DB".GC_MAN_SS;
      A     "HOOD_SYSTEM_DB".HOOD_STA_PB;
      O     "HOOD_SYSTEM_DB".WTR_PMP_MTR_ON_CMD;
      );
      A     "GUIDE_CAGE_DB".GC_TRA_FWD_LS;
      O;
      A     "GUIDE_CAGE_DB".GC_LOC_SS;
      A(;
      O     "HOOD_SYSTEM_DB".HOOD_STA_PB;
      O     "HOOD_SYSTEM_DB".WTR_PMP_MTR_ON_CMD;
      );
      );
      A     "HOOD_SYSTEM_DB".HOOD_STP_PB;
      AN    "HOOD_SYSTEM_DB".WTR_PMP_FLT;
      AN    "HOOD_SYSTEM_DB".WTR_PMP_MTR_TRIP_FB;
      A     "HOOD_SYSTEM_DB".WTR_PMP_MTR_RDY_FOR_STA;
      O;
      A     "ALWAYS_ON";
      A(;
      O     "GUIDE_CAGE_DB".GC_AUTO_SS;
      O     "GUIDE_CAGE_DB".GC_MAN_SS;
      );
      A     "GUIDE_CAGE_DB".GC_TRA_FWD_LS;
      A     "CMD_FROM_TATA".GC_OnBord_STATUS_BIT.HOOD_SYS_ON_CMD;
      AN    "HOOD_SYSTEM_DB".WTR_PMP_MTR_TRIP_FB;
      A     "HOOD_SYSTEM_DB".WTR_PMP_MTR_RDY_FOR_STA;
      );
      =     L 0.0;
      A     L 0.0;
      BLD   102;
      =     "HOOD_SYSTEM_DB".WTR_PMP_MTR_ON_CMD;
      A     L 0.0;
      FP    "HOOD_SYSTEM_DB".PULSE_1;
      JNB   _001;
      L     0;
      T     "HOOD_SYSTEM_DB".WTR_PMP_FLT_TMR;
_001: NOP   0;
      A     L 0.0;
      FN    "HOOD_SYSTEM_DB".PULSE_10;
      R     "HOOD_SYSTEM_DB".IDF_DRV_LOW_SPD_OVR;
NETWORK
TITLE = WATER PUMP MOTOR FAULT GENERATION
      A     "ALWAYS_ON";
      =     L 0.0;
      A     L 0.0;
      A     "HOOD_SYSTEM_DB".WTR_PMP_MTR_ON_CMD;
      AN    "HOOD_SYSTEM_DB".WTR_PMP_MTR_ON_FB;
      AN    "HOOD_SYSTEM_DB".WTR_PMP_FLT;
      A     "ONE_SECOND_PULSE";
      JNB   _002;
      L     1;
      L     "HOOD_SYSTEM_DB".WTR_PMP_FLT_TMR;
      +I;
      T     "HOOD_SYSTEM_DB".WTR_PMP_FLT_TMR;
_002: NOP   0;
      A     L 0.0;
      A(;
      L     "HOOD_SYSTEM_DB".WTR_PMP_FLT_TMR;
      L     "HOOD_SYSTEM_DB".WTR_PMP_FLT_GEN_TIME;
      >=I;
      );
      =     "AIR_COMPRESSOR_DB".AC_MTR_FLT;
      A     L 0.0;
      A     "MAIN_POWER_DB".ALARM_ACK_PB;
      A     "HOOD_SYSTEM_DB".WTR_PMP_FLT;
      JNB   _003;
      L     0;
      T     "HOOD_SYSTEM_DB".WTR_PMP_FLT_TMR;
_003: NOP   0;
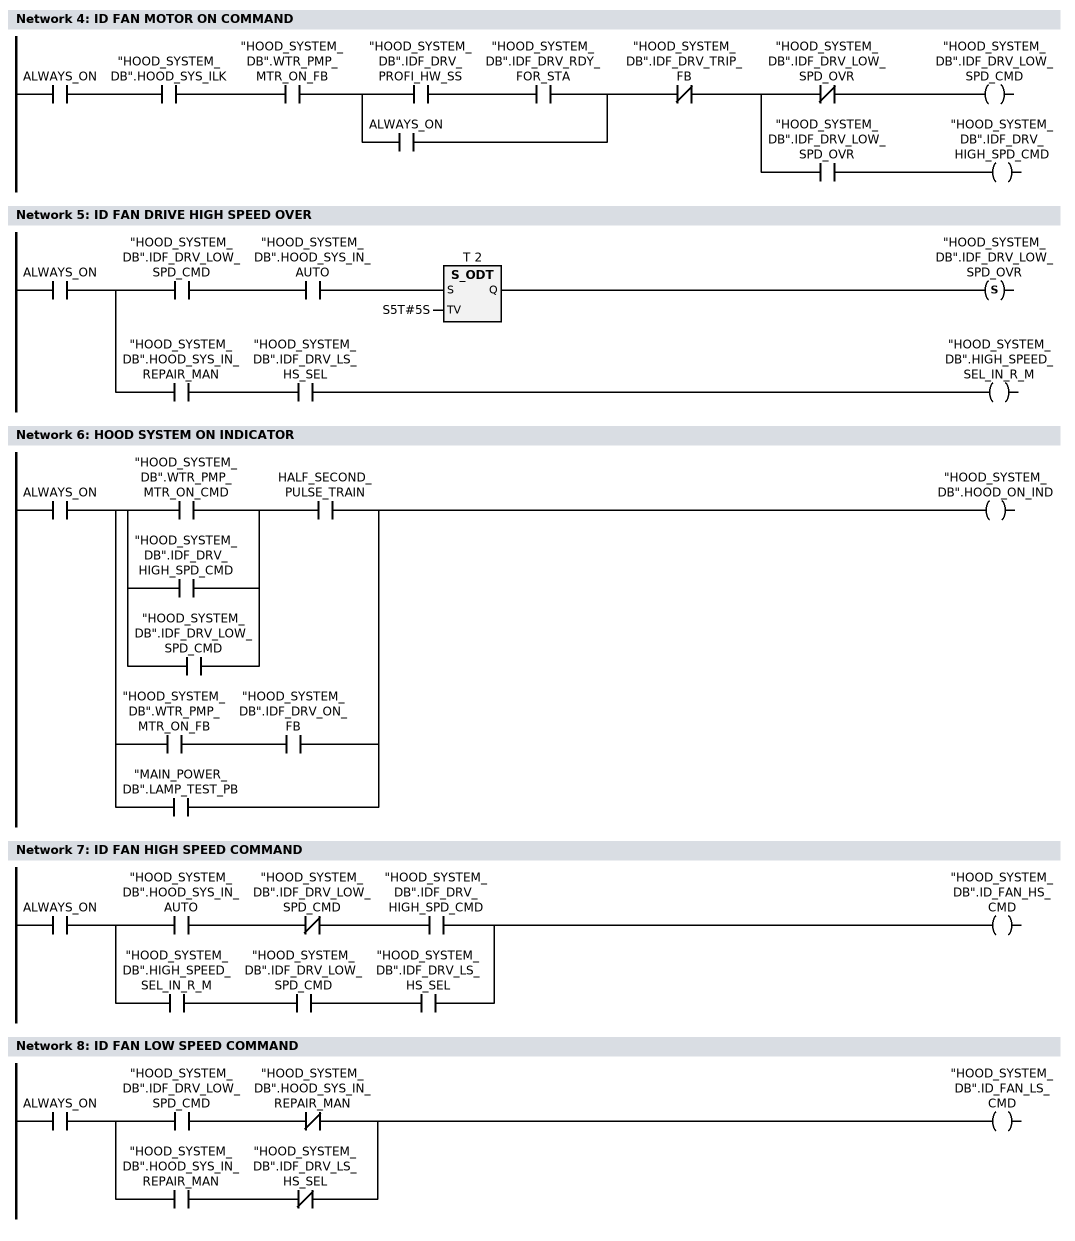
NETWORK
TITLE = ID FAN MOTOR ON COMMAND
      A     "ALWAYS_ON";
      A     "HOOD_SYSTEM_DB".HOOD_SYS_ILK;
      A     "HOOD_SYSTEM_DB".WTR_PMP_MTR_ON_FB;
      A(;
      A     "HOOD_SYSTEM_DB".IDF_DRV_PROFI_HW_SS;
      A     "HOOD_SYSTEM_DB".IDF_DRV_RDY_FOR_STA;
      O     "ALWAYS_ON";
      );
      AN    "HOOD_SYSTEM_DB".IDF_DRV_TRIP_FB;
      =     L 0.0;
      A     L 0.0;
      AN    "HOOD_SYSTEM_DB".IDF_DRV_LOW_SPD_OVR;
      =     "HOOD_SYSTEM_DB".IDF_DRV_LOW_SPD_CMD;
      A     L 0.0;
      A     "HOOD_SYSTEM_DB".IDF_DRV_LOW_SPD_OVR;
      =     "HOOD_SYSTEM_DB".IDF_DRV_HIGH_SPD_CMD;
NETWORK
TITLE = ID FAN DRIVE HIGH SPEED OVER
      A     "ALWAYS_ON";
      =     L 0.0;
      A     L 0.0;
      A     "HOOD_SYSTEM_DB".IDF_DRV_LOW_SPD_CMD;
      A     "HOOD_SYSTEM_DB".HOOD_SYS_IN_AUTO;
      L     S5T#5S;
      SD    T 2;
      NOP   0;
      NOP   0;
      NOP   0;
      A     T 2;
      S     "HOOD_SYSTEM_DB".IDF_DRV_LOW_SPD_OVR;
      A     L 0.0;
      A     "HOOD_SYSTEM_DB".HOOD_SYS_IN_REPAIR_MAN;
      A     "HOOD_SYSTEM_DB".IDF_DRV_LS_HS_SEL;
      =     "HOOD_SYSTEM_DB".HIGH_SPEED_SEL_IN_R_M;
NETWORK
TITLE = HOOD SYSTEM ON INDICATOR
      A     "ALWAYS_ON";
      A(;
      A(;
      O     "HOOD_SYSTEM_DB".WTR_PMP_MTR_ON_CMD;
      O     "HOOD_SYSTEM_DB".IDF_DRV_HIGH_SPD_CMD;
      O     "HOOD_SYSTEM_DB".IDF_DRV_LOW_SPD_CMD;
      );
      A     "HALF_SECOND_PULSE_TRAIN";
      O;
      A     "HOOD_SYSTEM_DB".WTR_PMP_MTR_ON_FB;
      A     "HOOD_SYSTEM_DB".IDF_DRV_ON_FB;
      O     "MAIN_POWER_DB".LAMP_TEST_PB;
      );
      =     "HOOD_SYSTEM_DB".HOOD_ON_IND;
NETWORK
TITLE = ID FAN HIGH SPEED COMMAND
      A     "ALWAYS_ON";
      A(;
      A     "HOOD_SYSTEM_DB".HOOD_SYS_IN_AUTO;
      AN    "HOOD_SYSTEM_DB".IDF_DRV_LOW_SPD_CMD;
      A     "HOOD_SYSTEM_DB".IDF_DRV_HIGH_SPD_CMD;
      O;
      A     "HOOD_SYSTEM_DB".HIGH_SPEED_SEL_IN_R_M;
      A     "HOOD_SYSTEM_DB".IDF_DRV_LOW_SPD_CMD;
      A     "HOOD_SYSTEM_DB".IDF_DRV_LS_HS_SEL;
      );
      =     "HOOD_SYSTEM_DB".ID_FAN_HS_CMD;
NETWORK
TITLE = ID FAN LOW SPEED COMMAND
      A     "ALWAYS_ON";
      A(;
      A     "HOOD_SYSTEM_DB".IDF_DRV_LOW_SPD_CMD;
      AN    "HOOD_SYSTEM_DB".HOOD_SYS_IN_REPAIR_MAN;
      O;
      A     "HOOD_SYSTEM_DB".HOOD_SYS_IN_REPAIR_MAN;
      AN    "HOOD_SYSTEM_DB".IDF_DRV_LS_HS_SEL;
      );
      =     "HOOD_SYSTEM_DB".ID_FAN_LS_CMD;
END_FUNCTION

FUNCTION "DOOR_EXTRACTOR" : VOID	// FC 8
TITLE = DOOR EXTRACTOR
AUTHOR : Kamillas
VERSION : 0.1
BEGIN
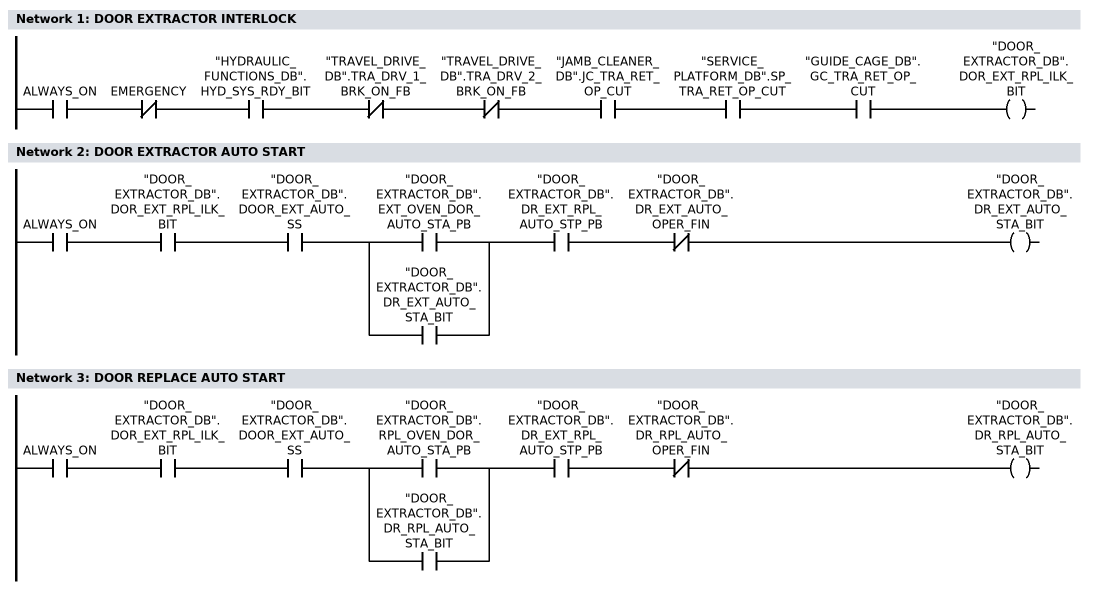
NETWORK
TITLE = DOOR EXTRACTOR INTERLOCK
      A     "ALWAYS_ON";
      AN    "EMERGENCY";
      A     "HYDRAULIC_FUNCTIONS_DB".HYD_SYS_RDY_BIT;
      AN    "TRAVEL_DRIVE_DB".TRA_DRV_1_BRK_ON_FB;
      AN    "TRAVEL_DRIVE_DB".TRA_DRV_2_BRK_ON_FB;
      A     "JAMB_CLEANER_DB".JC_TRA_RET_OP_CUT;
      A     "SERVICE_PLATFORM_DB".SP_TRA_RET_OP_CUT;
      A     "GUIDE_CAGE_DB".GC_TRA_RET_OP_CUT;
      =     "DOOR_EXTRACTOR_DB".DOR_EXT_RPL_ILK_BIT;
NETWORK
TITLE = DOOR EXTRACTOR AUTO START
      A     "ALWAYS_ON";
      A     "DOOR_EXTRACTOR_DB".DOR_EXT_RPL_ILK_BIT;
      A     "DOOR_EXTRACTOR_DB".DOOR_EXT_AUTO_SS;
      A(;
      O     "DOOR_EXTRACTOR_DB".EXT_OVEN_DOR_AUTO_STA_PB;
      O     "DOOR_EXTRACTOR_DB".DR_EXT_AUTO_STA_BIT;
      );
      A     "DOOR_EXTRACTOR_DB".DR_EXT_RPL_AUTO_STP_PB;
      AN    "DOOR_EXTRACTOR_DB".DR_EXT_AUTO_OPER_FIN;
      =     "DOOR_EXTRACTOR_DB".DR_EXT_AUTO_STA_BIT;
NETWORK
TITLE = DOOR REPLACE AUTO START
      A     "ALWAYS_ON";
      A     "DOOR_EXTRACTOR_DB".DOR_EXT_RPL_ILK_BIT;
      A     "DOOR_EXTRACTOR_DB".DOOR_EXT_AUTO_SS;
      A(;
      O     "DOOR_EXTRACTOR_DB".RPL_OVEN_DOR_AUTO_STA_PB;
      O     "DOOR_EXTRACTOR_DB".DR_RPL_AUTO_STA_BIT;
      );
      A     "DOOR_EXTRACTOR_DB".DR_EXT_RPL_AUTO_STP_PB;
      AN    "DOOR_EXTRACTOR_DB".DR_RPL_AUTO_OPER_FIN;
      =     "DOOR_EXTRACTOR_DB".DR_RPL_AUTO_STA_BIT;
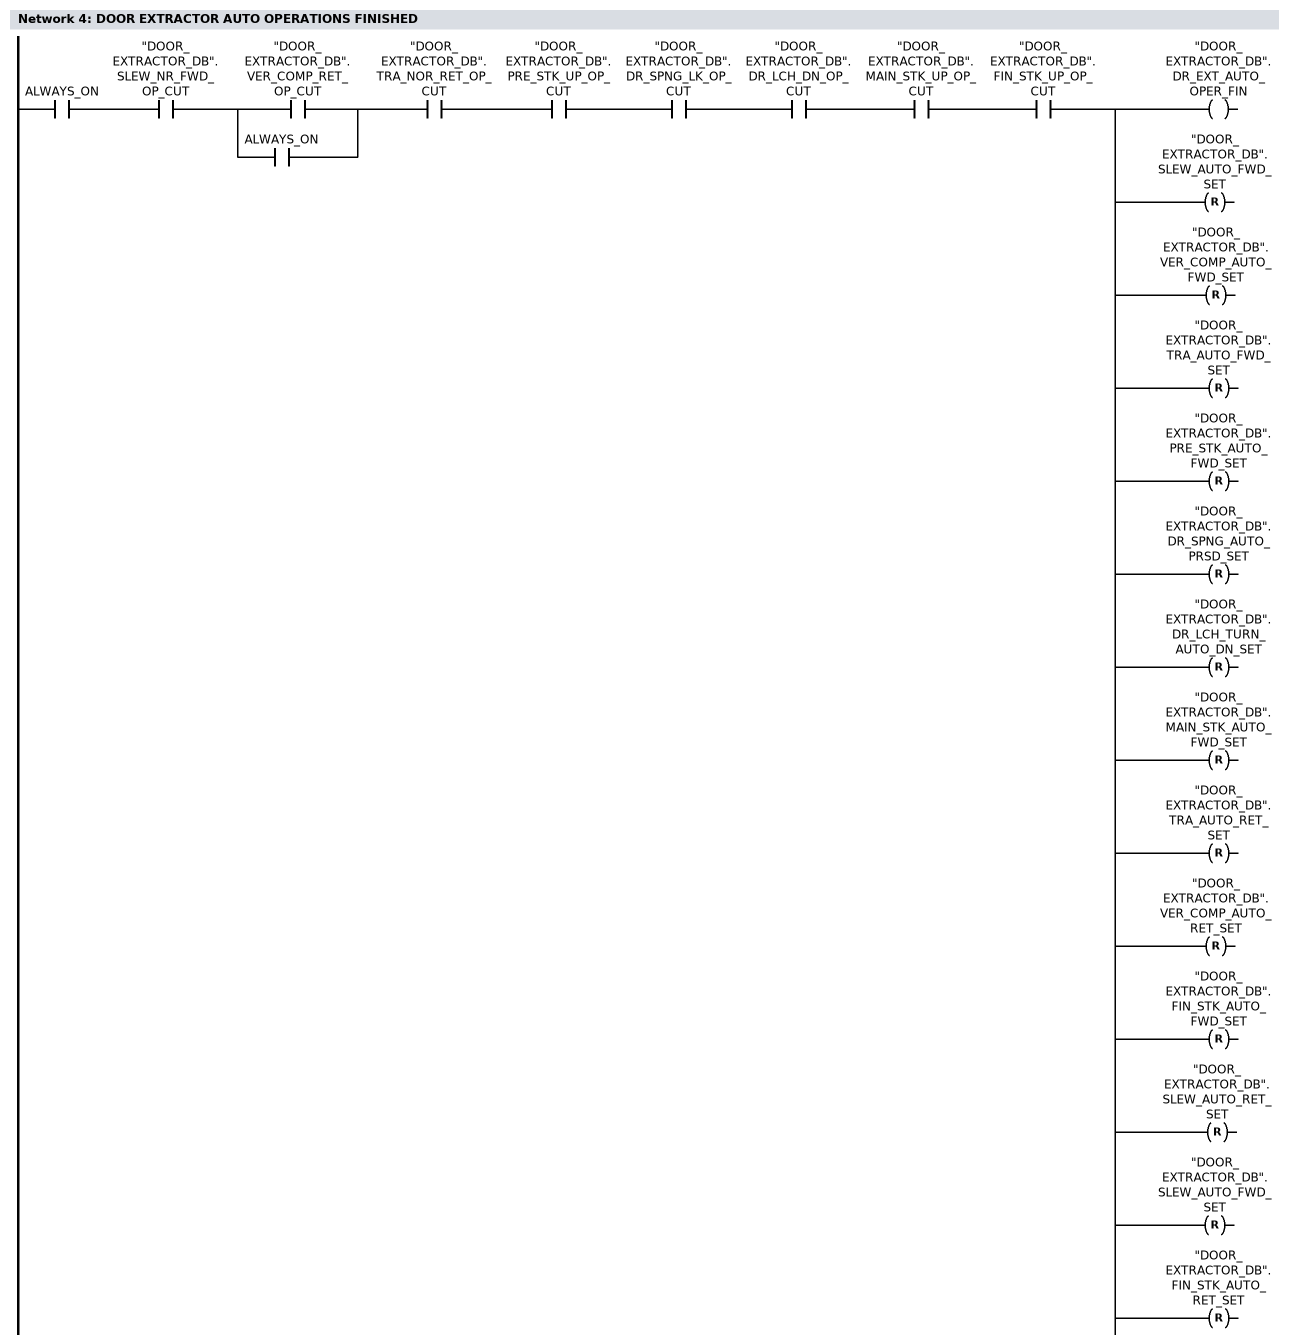
